(* Logix 5000 project; controller Amvex_Thorpe_Flowmeter vendor 1 type 14 code 106 rev 33.13; software revision 33.01; part 9 of 16 *)

ADD_ON_INSTRUCTION SetVelControlTimeOut   (* revision 0.1, vendor Mecademic Inc., ExecuteEnableInFalse *)
// Timeout for current velocity mode
VAR_IN_OUT
   RobotInputs : _061D:Meca500_86BDA20B:I:0; {required}
   RobotOutputs : _061D:Meca500_01F88326:O:0; {required}
END_VAR
VAR_INPUT
   Parameter_Value : REAL; {required}
   ExternalStateControl : BOOL; {required}
   ExternalMoveID : INT; {required}
END_VAR
VAR_OUTPUT
   Enabled : BOOL; {visible}
   Sent : BOOL; {visible}
   Buffered : BOOL; {visible}
   Error : BOOL; {visible}
END_VAR
VAR
   InternalMoveID : INT; {access None}
   MoveIDTrig : BOOL; {access None}
   MoveIDUpdated : BOOL; {access None}
   OneShot : DINT; {access None}
   FirstScan : BOOL; {access None}
END_VAR

ROUTINE EnableInFalse   (* ladder *)
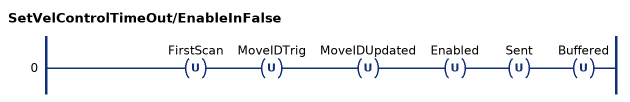
   0: OTU(FirstScan)OTU(MoveIDTrig)OTU(MoveIDUpdated)OTU(Enabled)OTU(Sent)OTU(Buffered);
END_ROUTINE

ROUTINE Logic   (* ladder *)
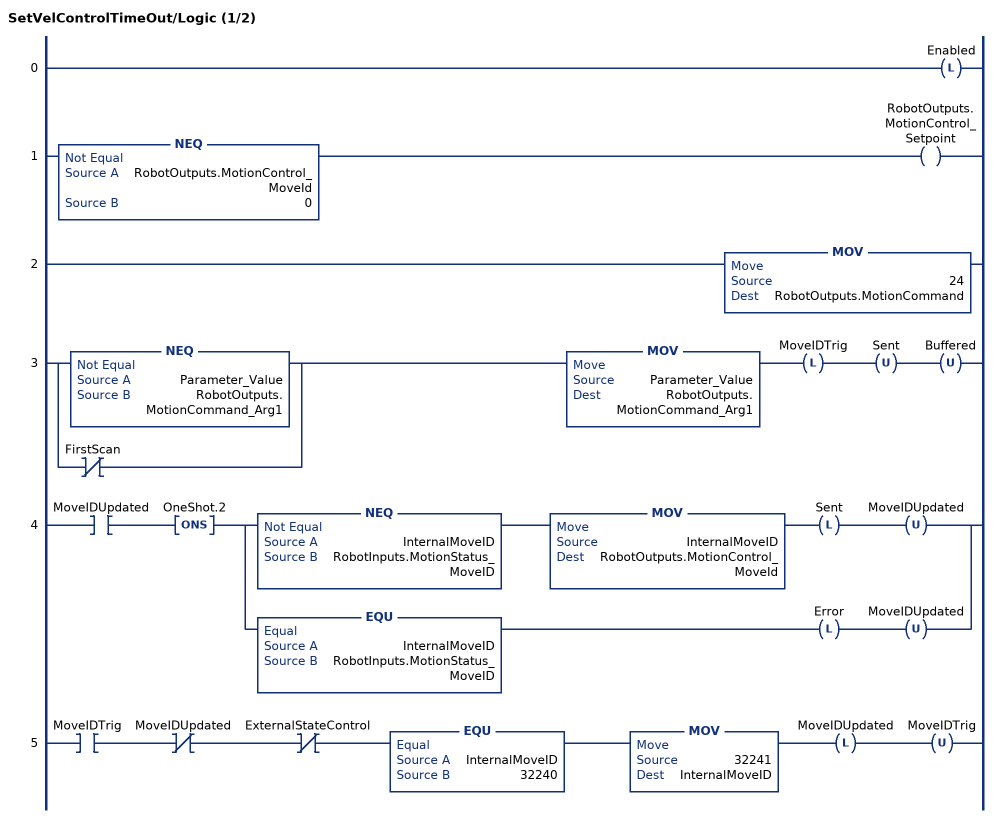
   0: OTL(Enabled);
   1: NEQ(RobotOutputs.MotionControl_MoveId,0)OTE(RobotOutputs.MotionControl_Setpoint);
   2: MOV(24,RobotOutputs.MotionCommand);
   3: [NEQ(Parameter_Value,RobotOutputs.MotionCommand_Arg1) ,XIO(FirstScan) ]MOV(Parameter_Value,RobotOutputs.MotionCommand_Arg1)OTL(MoveIDTrig)OTU(Sent)OTU(Buffered);
   4: XIC(MoveIDUpdated)ONS(OneShot.2)[NEQ(InternalMoveID,RobotInputs.MotionStatus_MoveID) MOV(InternalMoveID,RobotOutputs.MotionControl_MoveId) OTL(Sent) OTU(MoveIDUpdated) ,EQU(InternalMoveID,RobotInputs.MotionStatus_MoveID) OTL(Error) OTU(MoveIDUpdated) ];
   5: XIC(MoveIDTrig)XIO(MoveIDUpdated)XIO(ExternalStateControl)EQU(InternalMoveID,32240)MOV(32241,InternalMoveID)OTL(MoveIDUpdated)OTU(MoveIDTrig);
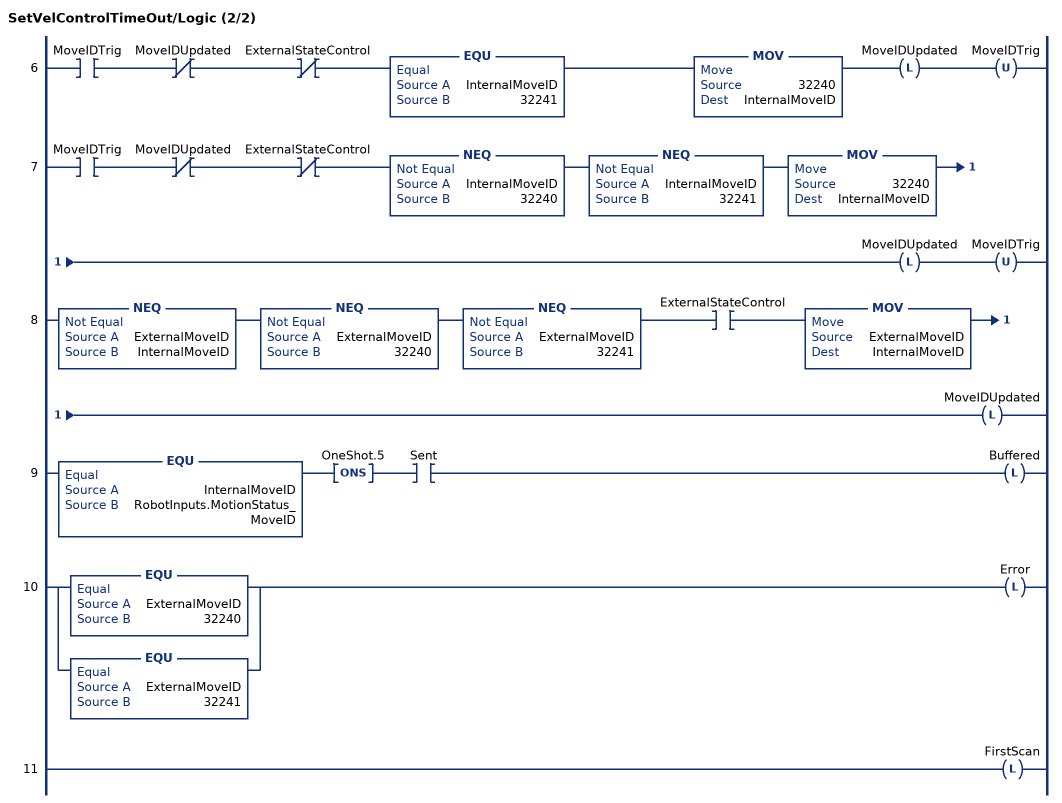
   6: XIC(MoveIDTrig)XIO(MoveIDUpdated)XIO(ExternalStateControl)EQU(InternalMoveID,32241)MOV(32240,InternalMoveID)OTL(MoveIDUpdated)OTU(MoveIDTrig);
   7: XIC(MoveIDTrig)XIO(MoveIDUpdated)XIO(ExternalStateControl)NEQ(InternalMoveID,32240)NEQ(InternalMoveID,32241)MOV(32240,InternalMoveID)OTL(MoveIDUpdated)OTU(MoveIDTrig);
   8: NEQ(ExternalMoveID,InternalMoveID)NEQ(ExternalMoveID,32240)NEQ(ExternalMoveID,32241)XIC(ExternalStateControl)MOV(ExternalMoveID,InternalMoveID)OTL(MoveIDUpdated);
   9: EQU(InternalMoveID,RobotInputs.MotionStatus_MoveID)ONS(OneShot.5)XIC(Sent)OTL(Buffered);
   10: [EQU(ExternalMoveID,32240) ,EQU(ExternalMoveID,32241) ]OTL(Error);
   11: OTL(FirstScan);
END_ROUTINE
END_ADD_ON_INSTRUCTION

ADD_ON_INSTRUCTION SetWRF   (* revision 0.1, vendor Mecademic Inc., ExecuteEnableInFalse *)
// Set the pose of the WRF with respect of the BRF
VAR_IN_OUT
   RobotInputs : _061D:Meca500_86BDA20B:I:0; {required}
   RobotOutputs : _061D:Meca500_01F88326:O:0; {required}
END_VAR
VAR_INPUT
   Pose_X_Pos : REAL; {required}
   Pose_Y_Pos : REAL; {required}
   Pose_Z_Pos : REAL; {required}
   Pose_rX_Ang : REAL; {required}
   Pose_rY_Ang : REAL; {required}
   Pose_rZ_Ang : REAL; {required}
   ExternalStateControl : BOOL; {required}
   ExternalMoveID : INT; {required}
END_VAR
VAR_OUTPUT
   Enabled : BOOL; {visible}
   Sent : BOOL; {visible}
   Buffered : BOOL; {visible}
   Error : BOOL; {visible}
END_VAR
VAR
   InternalMoveID : INT; {access None}
   MoveIDTrig : BOOL; {access None}
   MoveIDUpdated : BOOL; {access None}
   OneShot : DINT; {access None}
   FirstScan : BOOL; {access None}
END_VAR

ROUTINE EnableInFalse   (* ladder *)
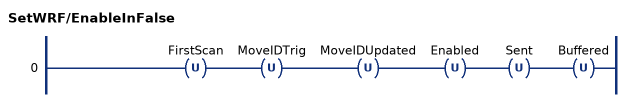
   0: OTU(FirstScan)OTU(MoveIDTrig)OTU(MoveIDUpdated)OTU(Enabled)OTU(Sent)OTU(Buffered);
END_ROUTINE

ROUTINE Logic   (* ladder *)
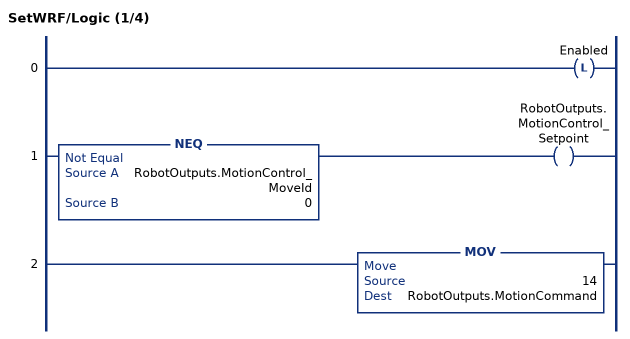
   0: OTL(Enabled);
   1: NEQ(RobotOutputs.MotionControl_MoveId,0)OTE(RobotOutputs.MotionControl_Setpoint);
   2: MOV(14,RobotOutputs.MotionCommand);
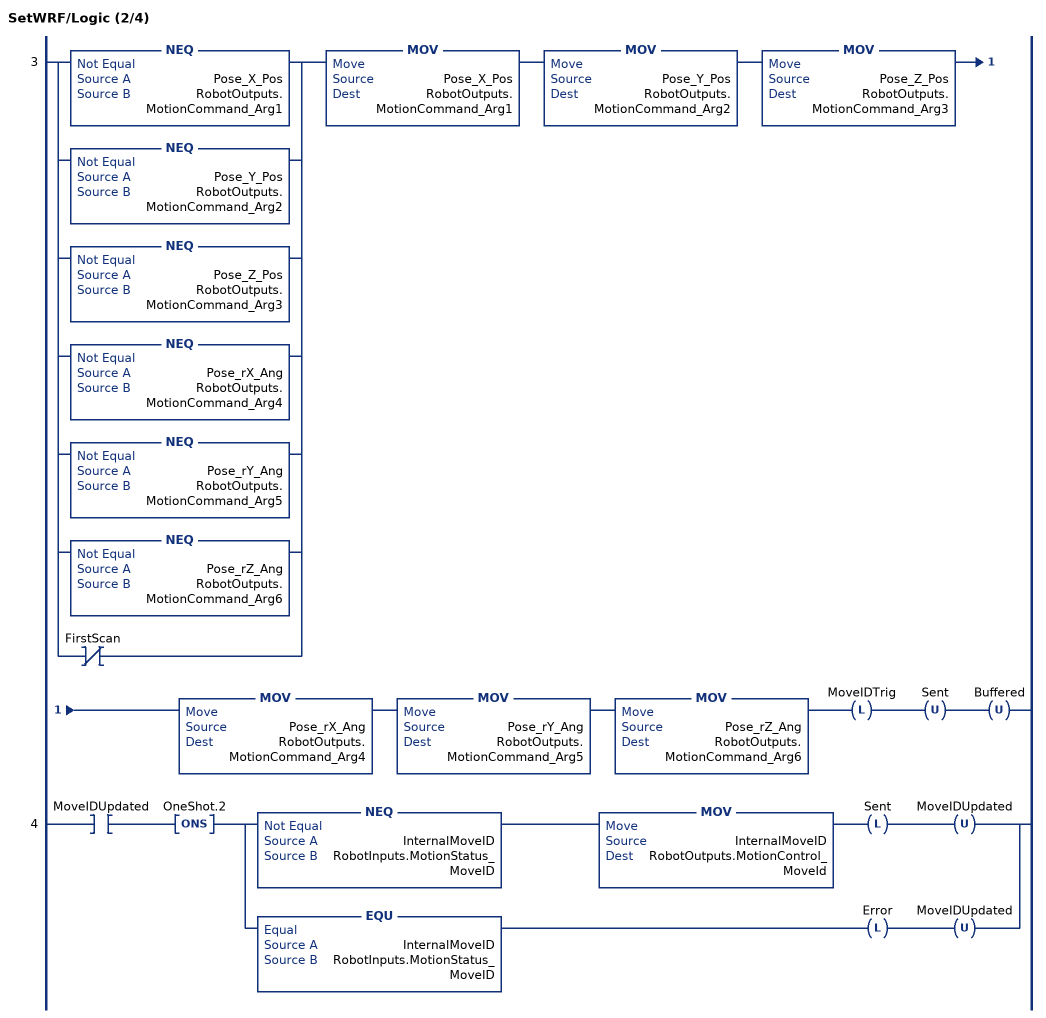
   3: [NEQ(Pose_X_Pos,RobotOutputs.MotionCommand_Arg1) ,NEQ(Pose_Y_Pos,RobotOutputs.MotionCommand_Arg2) ,NEQ(Pose_Z_Pos,RobotOutputs.MotionCommand_Arg3) ,NEQ(Pose_rX_Ang,RobotOutputs.MotionCommand_Arg4) ,NEQ(Pose_rY_Ang,RobotOutputs.MotionCommand_Arg5) ,NEQ(Pose_rZ_Ang,RobotOutputs.MotionCommand_Arg6) ,XIO(FirstScan) ]MOV(Pose_X_Pos,RobotOutputs.MotionCommand_Arg1)MOV(Pose_Y_Pos,RobotOutputs.MotionCommand_Arg2)MOV(Pose_Z_Pos,RobotOutputs.MotionCommand_Arg3)MOV(Pose_rX_Ang,RobotOutputs.MotionCommand_Arg4)MOV(Pose_rY_Ang,RobotOutputs.MotionCommand_Arg5)MOV(Pose_rZ_Ang,RobotOutputs.MotionCommand_Arg6)OTL(MoveIDTrig)OTU(Sent)OTU(Buffered);
   4: XIC(MoveIDUpdated)ONS(OneShot.2)[NEQ(InternalMoveID,RobotInputs.MotionStatus_MoveID) MOV(InternalMoveID,RobotOutputs.MotionControl_MoveId) OTL(Sent) OTU(MoveIDUpdated) ,EQU(InternalMoveID,RobotInputs.MotionStatus_MoveID) OTL(Error) OTU(MoveIDUpdated) ];
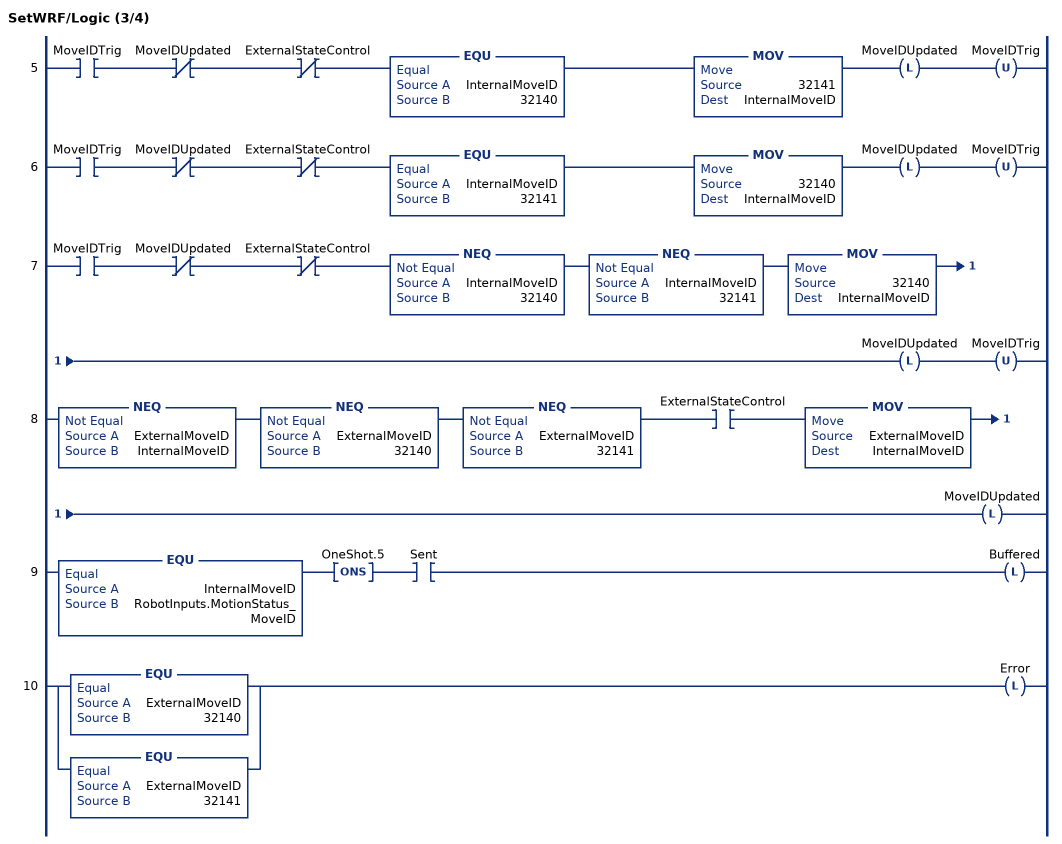
   5: XIC(MoveIDTrig)XIO(MoveIDUpdated)XIO(ExternalStateControl)EQU(InternalMoveID,32140)MOV(32141,InternalMoveID)OTL(MoveIDUpdated)OTU(MoveIDTrig);
   6: XIC(MoveIDTrig)XIO(MoveIDUpdated)XIO(ExternalStateControl)EQU(InternalMoveID,32141)MOV(32140,InternalMoveID)OTL(MoveIDUpdated)OTU(MoveIDTrig);
   7: XIC(MoveIDTrig)XIO(MoveIDUpdated)XIO(ExternalStateControl)NEQ(InternalMoveID,32140)NEQ(InternalMoveID,32141)MOV(32140,InternalMoveID)OTL(MoveIDUpdated)OTU(MoveIDTrig);
   8: NEQ(ExternalMoveID,InternalMoveID)NEQ(ExternalMoveID,32140)NEQ(ExternalMoveID,32141)XIC(ExternalStateControl)MOV(ExternalMoveID,InternalMoveID)OTL(MoveIDUpdated);
   9: EQU(InternalMoveID,RobotInputs.MotionStatus_MoveID)ONS(OneShot.5)XIC(Sent)OTL(Buffered);
   10: [EQU(ExternalMoveID,32140) ,EQU(ExternalMoveID,32141) ]OTL(Error);
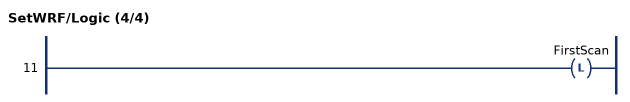
   11: OTL(FirstScan);
END_ROUTINE
END_ADD_ON_INSTRUCTION

ADD_ON_INSTRUCTION StartOfflineProgram   (* revision 0.1, vendor Mecademic Inc., ExecuteEnableInFalse *)
// Start an offline program with specified id
VAR_IN_OUT
   RobotInputs : _061D:Meca500_86BDA20B:I:0; {required}
   RobotOutputs : _061D:Meca500_01F88326:O:0; {required}
END_VAR
VAR_INPUT
   Parameter_Value : REAL; {required}
   ExternalStateControl : BOOL; {required}
   ExternalMoveID : INT; {required}
END_VAR
VAR_OUTPUT
   Enabled : BOOL; {visible}
   Sent : BOOL; {visible}
   Buffered : BOOL; {visible}
   Error : BOOL; {visible}
END_VAR
VAR
   InternalMoveID : INT; {access None}
   MoveIDTrig : BOOL; {access None}
   MoveIDUpdated : BOOL; {access None}
   OneShot : DINT; {access None}
   FirstScan : BOOL; {access None}
END_VAR

ROUTINE EnableInFalse   (* ladder *)
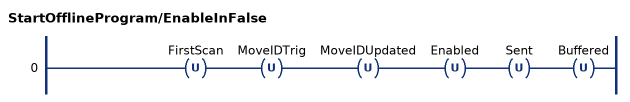
   0: OTU(FirstScan)OTU(MoveIDTrig)OTU(MoveIDUpdated)OTU(Enabled)OTU(Sent)OTU(Buffered);
END_ROUTINE

ROUTINE Logic   (* ladder *)
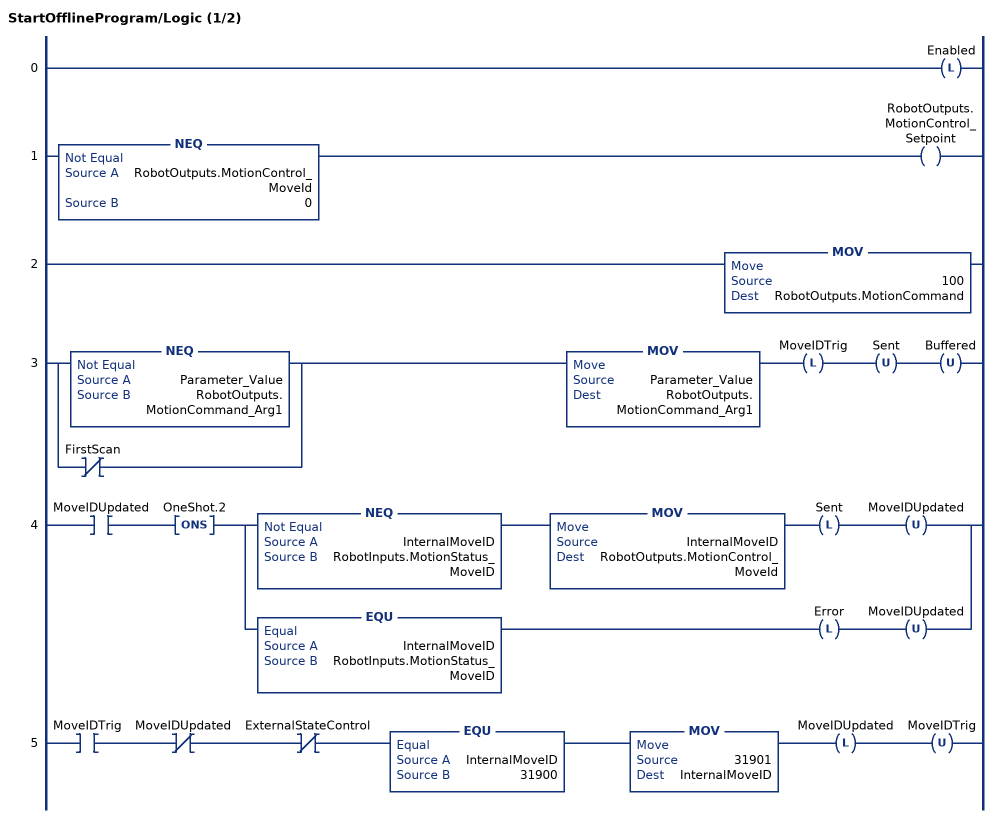
   0: OTL(Enabled);
   1: NEQ(RobotOutputs.MotionControl_MoveId,0)OTE(RobotOutputs.MotionControl_Setpoint);
   2: MOV(100,RobotOutputs.MotionCommand);
   3: [NEQ(Parameter_Value,RobotOutputs.MotionCommand_Arg1) ,XIO(FirstScan) ]MOV(Parameter_Value,RobotOutputs.MotionCommand_Arg1)OTL(MoveIDTrig)OTU(Sent)OTU(Buffered);
   4: XIC(MoveIDUpdated)ONS(OneShot.2)[NEQ(InternalMoveID,RobotInputs.MotionStatus_MoveID) MOV(InternalMoveID,RobotOutputs.MotionControl_MoveId) OTL(Sent) OTU(MoveIDUpdated) ,EQU(InternalMoveID,RobotInputs.MotionStatus_MoveID) OTL(Error) OTU(MoveIDUpdated) ];
   5: XIC(MoveIDTrig)XIO(MoveIDUpdated)XIO(ExternalStateControl)EQU(InternalMoveID,31900)MOV(31901,InternalMoveID)OTL(MoveIDUpdated)OTU(MoveIDTrig);
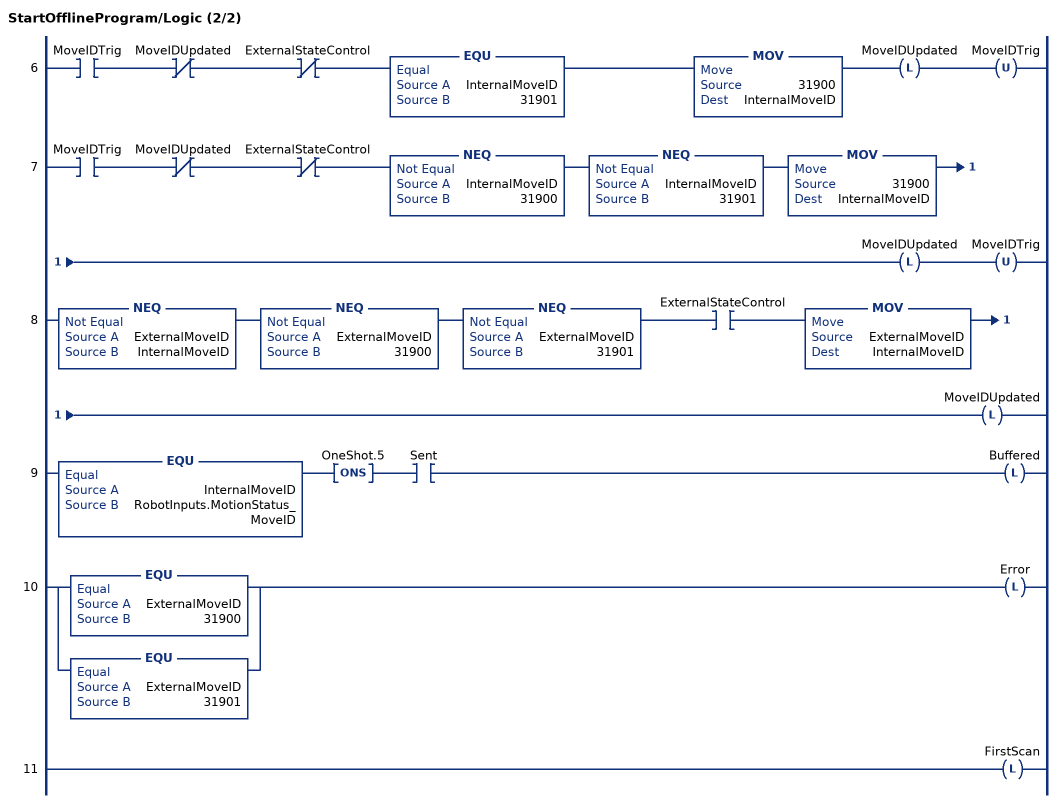
   6: XIC(MoveIDTrig)XIO(MoveIDUpdated)XIO(ExternalStateControl)EQU(InternalMoveID,31901)MOV(31900,InternalMoveID)OTL(MoveIDUpdated)OTU(MoveIDTrig);
   7: XIC(MoveIDTrig)XIO(MoveIDUpdated)XIO(ExternalStateControl)NEQ(InternalMoveID,31900)NEQ(InternalMoveID,31901)MOV(31900,InternalMoveID)OTL(MoveIDUpdated)OTU(MoveIDTrig);
   8: NEQ(ExternalMoveID,InternalMoveID)NEQ(ExternalMoveID,31900)NEQ(ExternalMoveID,31901)XIC(ExternalStateControl)MOV(ExternalMoveID,InternalMoveID)OTL(MoveIDUpdated);
   9: EQU(InternalMoveID,RobotInputs.MotionStatus_MoveID)ONS(OneShot.5)XIC(Sent)OTL(Buffered);
   10: [EQU(ExternalMoveID,31900) ,EQU(ExternalMoveID,31901) ]OTL(Error);
   11: OTL(FirstScan);
END_ROUTINE
END_ADD_ON_INSTRUCTION

VAR_GLOBAL   (* controller tags *)
   Air_Pressure_Issue_Delay_TMR : TIMER := (PRE := 1000, ACC := 1000, EN := 1, DN := 1);
   Alicat1RequestMsg : MESSAGE;
        MessageParameters(ServiceCode := 16#0010, LocalElement := MCP.Testing.Alicat[0].CmdData[0], ...)
   Alicat1ResponseMsg : MESSAGE;
        MessageParameters(ServiceCode := 16#000e, DestinationTag := MCP.Testing.Alicat[0].CmdData[0], ...)
   Alicat2RequestMsg : MESSAGE;
        MessageParameters(ServiceCode := 16#0010, LocalElement := MCP.Testing.Alicat[1].CmdData[0], ...)
   Alicat2ResponseMsg : MESSAGE;
        MessageParameters(ServiceCode := 16#000e, DestinationTag := MCP.Testing.Alicat[1].CmdData[0], ...)
   Alicat5LPM_Timeout : TIMER := (PRE := 3000);
   Alicat_Status_ONS : BOOL[32];
   Barcode_Data_String : STRING := '62810150300021T15UOB00032$0D$00$00$00$00$00$00$00$00$00$00$00$00$00$00$00$00$00$00$00$00$00$00$00$00$00$00$00$00$00$00$00$00$00$00$00$00$00$00$00$00$00$00$00$00$00$00$00$00$00$00$00$00$00$00$00$00$00$00';
   Barcode_Data_Temp : DINT;
   Barcode_Delay : TIMER := (PRE := 500);
   Barcode_timeout : TIMER := (PRE := 2000);
   Blank_Nest_Release_TMR : TIMER := (PRE := 500);
   Close : BOOL;
   Close_Go_ONS : BOOL;
   Close_Knob : Servo_Move := (Speed := 400.0, Torque := 37.0, Position := 100000.0, Path := 1);
   Close_Knob_Step : Servo_Move := (Speed := 600.0, Torque := 35.0, Position := -100000.0, Path := 1);
   Close_ONS : BOOL;
   Close_Rapid : Servo_Move := (Speed := 8000.0, Torque := 80.0, Position := 550000.0, Path := 1);
   Close_Step : Servo_Move := (Speed := 600.0, Torque := 37.0, Position := 1000000.0, Path := 1);
   Close_Stop : BOOL;
   Close_Torque : INT := 36;
   Close_Torque_TMR : TIMER;
   CloseKnob : Servo_Move := (Speed := 200.0, Torque := 55.0, Position := 1000000.0, Path := 1);
   Cycle_Count_Ctr : COUNTER := (ACC := 1765, DN := 1);
   Cycle_Count_ONS : BOOL;
   Cycle_Time_ONS : BOOL;
   Cycle_Timer_ONS : BOOL;
   Datalogging_Time_Delay : TIMER := (PRE := 500);
   Delay : TIMER := (PRE := 3000);
   Downsteam_Release_ONS1 : BOOL;
   Downsteam_Release_ONS2 : BOOL;
   Empty_Pallet_Timer : TIMER := (PRE := 5000);
   Empty_Pallet_Timer2 : TIMER := (PRE := 5000);
   End_Of_Cycle : BOOL;
   Fastest_Delay : TIMER := (PRE := 100);
   FIRST_SCAN : BOOL;
   FIRST_SCAN_ONS : BOOL := 1;
   Fitting_Cycle_Timer : TIMER := (PRE := 6000000);
   Fitting_Cycle_Timer_DINT : DINT;
   Fitting_Cycle_Timer_ONS : BOOL;
   Flood_delay : TIMER := (PRE := 10000, ACC := 10000, EN := 1, DN := 1);
   Flowmeter_Record : STRING;
   HMI : HMI_Temp;
   ID0_InputDataLength : MESSAGE;   // Message Command Input Data Data Length
        MessageParameters(ServiceCode := 16#000e, DestinationTag := RCP1_00.MISC.InputBytes, ...)
   ID0_LengthParameterdata : MESSAGE;   // Message Command Parameter Data Length
        MessageParameters(ServiceCode := 16#000e, DestinationTag := RCP1_00.MISC.ParameterBytes, ...)
   ID0_MSG_Diagnostic : MESSAGE;   // Message Get Diagnosis Module
        MessageParameters(ServiceCode := 16#000e, DestinationTag := RCP1_00.MISC.DiagnosticData[0], ...)
   ID0_MSG_ProcessAlarm : MESSAGE;   // Message Get Get Process Alram Module
        MessageParameters(ServiceCode := 16#000e, DestinationTag := RCP1_00.MISC.ProcessAlarmData[0], ...)
   ID0_OutputDataLength : MESSAGE;   // Message Command Output Data Data Length
        MessageParameters(ServiceCode := 16#000e, DestinationTag := RCP1_00.MISC.OutputBytes, ...)
   ID0_ReceiveMSG1 : MESSAGE;   // Message Command Parameter Receive Data
        MessageParameters(ServiceCode := 16#000e, DestinationTag := RCP1_00.MISC.ParameterArray_RX_TX[0], ...)
   ID0_ReceiveMSG2 : MESSAGE;   // Message Command Parameter Receive Data
        MessageParameters(ServiceCode := 16#000e, DestinationTag := RCP1_00.MISC.ParameterArray_RX_TX[450], ...)
   ID0_ReceiveMSG3 : MESSAGE;   // Message Command Parameter Receive Data
        MessageParameters(ServiceCode := 16#000e, DestinationTag := RCP1_00.MISC.ParameterArray_RX_TX[900], ...)
   ID0_SendMSG1 : MESSAGE;   // Message Command Parameter Send Data
        MessageParameters(ServiceCode := 16#0010, LocalElement := RCP1_00.MISC.ParameterArray_RX_TX[0], ...)
   ID0_SendMSG2 : MESSAGE;   // Message Command Parameter Send Data
        MessageParameters(ServiceCode := 16#0010, LocalElement := RCP1_00.MISC.ParameterArray_RX_TX[450], ...)
   ID0_SendMSG3 : MESSAGE;   // Message Command Parameter Send Data
        MessageParameters(ServiceCode := 16#0010, LocalElement := RCP1_00.MISC.ParameterArray_RX_TX[900], ...)
   ID86_InputDataLength : MESSAGE;   // Message Command Input Data Data Length
        MessageParameters(ServiceCode := 16#000e, DestinationTag := MCP_00.MISC.InputBytes, ...)
   ID86_LengthParameterdata : MESSAGE;   // Message Command Parameter Data Length
        MessageParameters(ServiceCode := 16#000e, DestinationTag := MCP_00.MISC.ParameterBytes, ...)
   ID86_MSG_Diagnostic : MESSAGE;   // Message Get Diagnosis Module
        MessageParameters(ServiceCode := 16#000e, DestinationTag := MCP_00.MISC.DiagnosticData[0], ...)
   ID86_MSG_ProcessAlarm : MESSAGE;   // Message Get Get Process Alram Module
        MessageParameters(ServiceCode := 16#000e, DestinationTag := MCP_00.MISC.ProcessAlarmData[0], ...)
   ID86_OutputDataLength : MESSAGE;   // Message Command Output Data Data Length
        MessageParameters(ServiceCode := 16#000e, DestinationTag := MCP_00.MISC.OutputBytes, ...)
   ID86_ReceiveMSG1 : MESSAGE;   // Message Command Parameter Receive Data
        MessageParameters(ServiceCode := 16#000e, DestinationTag := MCP_00.MISC.ParameterArray_RX_TX[0], ...)
   ID86_ReceiveMSG2 : MESSAGE;   // Message Command Parameter Receive Data
        MessageParameters(ServiceCode := 16#000e, DestinationTag := MCP_00.MISC.ParameterArray_RX_TX[450], ...)
   ID86_ReceiveMSG3 : MESSAGE;   // Message Command Parameter Receive Data
        MessageParameters(ServiceCode := 16#000e, DestinationTag := MCP_00.MISC.ParameterArray_RX_TX[900], ...)
   ID86_SendMSG1 : MESSAGE;   // Message Command Parameter Send Data
        MessageParameters(ServiceCode := 16#0010, LocalElement := MCP_00.MISC.ParameterArray_RX_TX[0], ...)
   ID86_SendMSG2 : MESSAGE;   // Message Command Parameter Send Data
        MessageParameters(ServiceCode := 16#0010, LocalElement := MCP_00.MISC.ParameterArray_RX_TX[450], ...)
   ID86_SendMSG3 : MESSAGE;   // Message Command Parameter Send Data
        MessageParameters(ServiceCode := 16#0010, LocalElement := MCP_00.MISC.ParameterArray_RX_TX[900], ...)
   In_Cycle : BOOL := 1;
   Job_Number : STRING;
   KB_DeBug : DINT := 8424448;
   KB_Temp_Ret_TM : TIMER := (PRE := 600, ACC := 600, EN := 1, DN := 1);
   Knob_Closer : Servo_Move := (Speed := 600.0, Torque := 37.0, Position := -100000.0, Path := 1);
   Knob_Servo_Reset : BOOL := 1;
   Knob_Temp_Seq_Start : BOOL;
   Knob_Turner_ONS : BOOL;
   Last_Test_Data : REAL[8] := ([1] := 0.0001953125, [2] := 6.9492188, [3] := 15.0859375, [4] := 52.21875, [5] := 0.0005859375);
   Load_PB_ONS : BOOL;
   MCP : MCP := (Conv.VFD.Speed := 400, Conv.VFD.Ready := 1, Conv.Stop[0].Present.INPUT := 1, Conv.Stop[0].Present.ON_TIME := 100.0, Conv.Stop[0].Present.OFF_TIME := 50.0, Conv.Stop[0].Present.DEB_INPUT := 1, Conv.Stop[0].Present.IN := 1, Conv.Stop[0].Present.OUT := 1, Conv.Stop[1].Present.ON_TIME := 50.0, Conv.Stop[1].Present.OFF_TIME := 50.0, Conv.Stop[2].Present.INPUT := 1, Conv.Stop[2].Present.ON_TIME := 100.0, Conv.Stop[2].Present.OFF_TIME := 50.0, Conv.Stop[2].Present.DEB_INPUT := 1, Conv.Stop[2].Present.IN := 1, Conv.Stop[2].Present.OUT := 1, Conv.Lift.Stop.Present.INPUT := 1, Conv.Lift.Stop.Present.ON_TIME := 100.0, Conv.Lift.Stop.Present.OFF_TIME := 50.0, Conv.Lift.Stop.Present.DEB_INPUT := 1, Conv.Lift.Stop.Present.IN := 1, Conv.Lift.Stop.Present.OUT := 1, Conv.Lift.Extd.INPUT := 1, Conv.Lift.Extd.ON_TIME := 100.0, Conv.Lift.Extd.OFF_TIME := 50.0, Conv.Lift.Extd.DEB_INPUT := 1, Conv.Lift.Extd.IN := 1, Conv.Lift.Extd.OUT := 1, Conv.Lift.Retd.ON_TIME := 100.0, Conv.Lift.Retd.OFF_TIME := 50.0, Conv.Drop_TM[0].PRE := 250, Conv.Downstream_Full.ON_TIME := 50.0, Conv.Downstream_Full.OFF_TIME := 1000.0, Conv.Reject_Full.INPUT := 1, Conv.Reject_Full.ON_TIME := 250.0, Conv.Reject_Full.OFF_TIME := 50.0, Conv.Reject_Full.DEB_INPUT := 1, Conv.Reject_Full.IN := 1, Conv.Reject_Full.OUT := 1, Testing.Robot.Connection.Connect := 1, Testing.Robot.Connection.ConnectionFailed := 1, Testing.Robot.Lin_Speed := 85.0, Testing.Robot.Turn_TM.PRE := 350, Testing.Robot.Turn_Speed := 75.0, Testing.Robot.Turn_ONS := 1, Testing.Robot.MoveLin_Pos[0] := 64.35501, Testing.Robot.MoveLin_Pos[1] := 90.0, Testing.Robot.MoveLin_Pos[2] := 358.12, Testing.Robot.MoveLin_Pos[3] := -90.128174, Testing.Robot.MoveLin_Pos[4] := 2.1866865e-07, Testing.Robot.MoveLin_Pos[5] := -29.132236, Testing.Robot.Tool_Position_1[0] := 64.35501, Testing.Robot.Tool_Position_1[1] := 90.0, Testing.Robot.Tool_Position_1[2] := 358.12, Testing.Robot.Tool_Position_1[3] := -90.128174, Testing.Robot.Tool_Position_1[4] := 2.1866865e-07, Testing.Robot.Tool_Position_1[5] := -29.132236, Testing.Robot.Tool_Position_2[0] := 64.355, Testing.Robot.Tool_Position_2[1] := 130.0, Testing.Robot.Tool_Position_2[2] := 358.12,
        Testing.Robot.Tool_Position_2[3] := -90.0, Testing.Robot.Tool_Position_2[4] := -4.4799222e-07, Testing.Robot.Tool_Position_2[5] := -34.710915, Testing.Robot.At_Pos_1 := 1, Testing.Robot.DN := 1, Testing.Robot.Knob_Torque := 50.0, Testing.Robot.Jog.Increment := 5.0, Testing.Robot.Turn_Speed_AOI.Parameter_Value := 75.0, Testing.Robot.Turn_AOI.Joint_1_Angle := 17.26414, Testing.Robot.Turn_AOI.Joint_2_Angle := -8.834411, Testing.Robot.Turn_AOI.Joint_3_Angle := -19.158821, Testing.Robot.Turn_AOI.Joint_4_Angle := -98.415184, Testing.Robot.Turn_AOI.Joint_5_Angle := -74.87032, Testing.Robot.Torque_Config_AOI.Severity := 2.0, Testing.Robot.Torque_Limit_AOI.Joint_1_Limit := 100.0, Testing.Robot.Torque_Limit_AOI.Joint_2_Limit := 100.0, Testing.Robot.Torque_Limit_AOI.Joint_3_Limit := 100.0, Testing.Robot.Torque_Limit_AOI.Joint_4_Limit := 100.0, Testing.Robot.Torque_Limit_AOI.Joint_5_Limit := 100.0, Testing.Robot.Torque_Limit_AOI.Joint_6_Limit := 50.0, Testing.Robot.MoveLin_AOI.Pose_X_Pos := 64.35501, Testing.Robot.MoveLin_AOI.Pose_Y_Pos := 90.0, Testing.Robot.MoveLin_AOI.Pose_Z_Pos := 358.12, Testing.Robot.MoveLin_AOI.Pose_rX_Ang := -90.128174, Testing.Robot.MoveLin_AOI.Pose_rY_Ang := 2.1866865e-07, Testing.Robot.MoveLin_AOI.Pose_rZ_Ang := -29.132236, Testing.Robot.LinVel_AOI.Parameter_Value := 85.0, Testing.Robot.Open := 1, Testing.FastTest.Extd.INPUT := 1, Testing.FastTest.Extd.ON_TIME := 100.0, Testing.FastTest.Extd.OFF_TIME := 50.0, Testing.FastTest.Extd.DEB_INPUT := 1, Testing.FastTest.Extd.IN := 1, Testing.FastTest.Extd.OUT := 1, Testing.FastTest.Retd.ON_TIME := 100.0, Testing.FastTest.Retd.OFF_TIME := 50.0, Testing.Hood.Extd.INPUT := 1, Testing.Hood.Extd.ON_TIME := 100.0, Testing.Hood.Extd.OFF_TIME := 50.0, Testing.Hood.Extd.DEB_INPUT := 1, Testing.Hood.Extd.IN := 1, Testing.Hood.Extd.OUT := 1, Testing.Hood.Retd.ON_TIME := 100.0, Testing.Hood.Retd.OFF_TIME := 50.0, Testing.Alicat[0].IoData.Pressure := 14.396875, Testing.Alicat[0].IoData.Temperature := 28.3375, Testing.Alicat[0].IoData.VolFlow := 0.0001953125, Testing.Alicat[0].IoData.MassFlow := 0.0001953125, Testing.Alicat[0].IoData.GasIndex := 11, Testing.Alicat[0].IoData.Config := 16#0f, Testing.Alicat[0].IoData.PRESS := 1, Testing.Alicat[0].IoData.TEMP := 1, Testing.Alicat[0].IoData.VFLOW := 1, Testing.Alicat[0].IoData.MFLOW := 1, Testing.Alicat[0].Oxygen.To_100LPM := 1, Testing.Alicat[0].Ready := 1, Testing.Alicat[0].Flow := 0.0001953125, Testing.Alicat[0].Flow_data[0] := 1.5392579, Testing.Alicat[0].Flow_data[1] := 1.5396484, Testing.Alicat[0].Flow_data[2] := 1.5369141,
        Testing.Alicat[0].Flow_data[3] := 1.5371094, Testing.Alicat[0].Flow_data[4] := 1.5373048, Testing.Alicat[0].Flow_data[5] := 1.5378907, Testing.Alicat[0].Flow_data[6] := 1.5378907, Testing.Alicat[0].Flow_data[7] := 1.5382813, Testing.Alicat[0].Flow_data[8] := 1.5386719, Testing.Alicat[0].Flow_data[9] := 1.5386719, Testing.Alicat[0].Flow_data[10] := 1.5388672, Testing.Alicat[0].Flow_TM1.PRE := 1000, Testing.Alicat[0].Flow_TM2.PRE := 75, Testing.Alicat[1].IoData.Pressure := 14.396094, Testing.Alicat[1].IoData.Temperature := 25.284376, Testing.Alicat[1].IoData.VolFlow := 0.00390625, Testing.Alicat[1].IoData.MassFlow := 0.00390625, Testing.Alicat[1].IoData.GasIndex := 11, Testing.Alicat[1].IoData.Config := 16#0f, Testing.Alicat[1].IoData.PRESS := 1, Testing.Alicat[1].IoData.TEMP := 1, Testing.Alicat[1].IoData.VFLOW := 1, Testing.Alicat[1].IoData.MFLOW := 1, Testing.Alicat[1].Ready := 1, Testing.Alicat[1].Flow := 0.00390625, Testing.Alicat[1].Flow_data[0] := 7.8242188, Testing.Alicat[1].Flow_data[1] := 7.8164062, Testing.Alicat[1].Flow_data[2] := 7.8085938, Testing.Alicat[1].Flow_data[3] := 7.8046875, Testing.Alicat[1].Flow_data[4] := 7.796875, Testing.Alicat[1].Flow_data[5] := 7.796875, Testing.Alicat[1].Flow_data[6] := 7.796875, Testing.Alicat[1].Flow_data[7] := 7.84375, Testing.Alicat[1].Flow_data[8] := 7.8476562, Testing.Alicat[1].Flow_data[9] := 7.8398438, Testing.Alicat[1].Flow_data[10] := 7.8320312, Testing.Alicat[1].Flow_TM1.PRE := 1000, Testing.Alicat[1].Flow_TM2.PRE := 75, Testing.Alicat[1].Upper_Lim_Num := 8.8, Testing.Alicat[1].Lower_Lim_Num := 7.2, Testing.Vision.Prog := 3, Testing.Vision.Current_Prog := 3, Testing.Vision.Trigger_ON_TM.PRE := 33, Testing.Vision.Trigger_OFF_TM.PRE := 33, Testing.Barcode.Ready := 1, Testing.Barcode.Result := '010062810150300021T15UOB00032$0D', Testing.Part_Present.ON_TIME := 500.0, Testing.Part_Present.OFF_TIME := 50.0, Testing.Saftey.Light_Curtain := 1, Testing.Saftey.Output := 1, Testing.Saftey.RDC_Code := 15332, Testing.Air_pressure.INPUT := 1, Testing.Air_pressure.ON_TIME := 100.0, Testing.Air_pressure.OFF_TIME := 50.0, Testing.Air_pressure.DEB_INPUT := 1, Testing.Air_pressure.IN := 1, Testing.Air_pressure.OUT := 1, Testing.Part[39].Code := '010062810150300021T15UOB35098$0D', Testing.Part[39].Results := 56, Testing.Test[1].Range := 0.1, Testing.Test[1].Test_TM.PRE := 500, Testing.Test[1].Time := 1000, Testing.Test[2].Flow := 2.0,
        Testing.Test[2].Range := 0.5, Testing.Test[2].Test_TM.PRE := 500, Testing.Test[2].Time := 50, Testing.Test[3].Flow := 8.0, Testing.Test[3].Range := 0.8, Testing.Test[3].Test_TM.PRE := 500, Testing.Test[3].Time := 1, Testing.Test[4].Flow := 15.0, Testing.Test[4].Range := 1.5, Testing.Test[4].Test_TM.PRE := 500, Testing.Test[4].Time := 4007, Testing.Test[5].Flow := 50.0, Testing.Test[5].Range := 20.0, Testing.Test[5].Test_TM.PRE := 500, Testing.Test[5].Time := 13, Testing.Test[6].Test_TM.PRE := 1000, Testing.Test[6].Time := 4884, Testing.Load_PB.ON_TIME := 50.0, Testing.Load_PB.OFF_TIME := 50.0, Testing.Knob_Turner.Enable := 1, Testing.Knob_Turner.Stop := 1, Testing.Knob_Turner.Turn_Speed := 50.0, Testing.Knob_Turner.Rapid_Speed := 600.0, Testing.Knob_Turner.T2_Rapid_Pos := 550000.0, Testing.Knob_Turner.Torque_EN1 := 1, Testing.Knob_Turner.Torque_Feedback := 3.0, Testing.Knob_Turner.Path := 1.0, Testing.Knob_Turner.Extd.INPUT := 1, Testing.Knob_Turner.Extd.ON_TIME := 50.0, Testing.Knob_Turner.Extd.OFF_TIME := 50.0, Testing.Knob_Turner.Extd.DEB_INPUT := 1, Testing.Knob_Turner.Extd.IN := 1, Testing.Knob_Turner.Extd.OUT := 1, Testing.Knob_Turner.Retd.ON_TIME := 100.0, Testing.Knob_Turner.Retd.OFF_TIME := 50.0, Part_Count := 98, Lifetime_Part_Count := 5720.0, Fault_AOI[0].Timer_PRE := 2500, Fault_AOI[1].Timer_PRE := 2500, Fault_AOI[2].Timer_PRE := 2500, Fault_AOI[3].Timer_PRE := 2500, Fault_AOI[4].Timer_PRE := 2500, Fault_AOI[5].Timer_PRE := 2500, Fault_AOI[6].Timer_PRE := 2500, Fault_AOI[7].Timer_PRE := 2500, Fault_AOI[8].Timer_PRE := 2500, Fault_AOI[9].Timer_PRE := 2500, Fault_AOI[10].Timer_PRE := 2500, Fault_AOI[11].Timer_PRE := 2500, Fault_AOI[12].Timer_PRE := 2500, Fault_AOI[13].Timer_PRE := 2500, Fault_AOI[14].Timer_PRE := 2500, Fault_AOI[15].Timer_PRE := 2500, Fault_AOI[16].Timer_PRE := 2500, Fault_AOI[17].Timer_PRE := 2500, Fault_AOI[18].Timer_PRE := 2500, Fault_AOI[19].Timer_PRE := 2500, Fault_AOI[20].Timer_PRE := 2500, Fault_AOI[21].Fault := 1, Fault_AOI[21].Bypass := 1,
        Fault_AOI[21].Timer_PRE := 13, Fault_AOI[21].Faulted := 1, Fault_AOI[22].Fault := 1, Fault_AOI[22].Timer_PRE := 63968020, Fault_AOI[22].Timer_ACC := 4079810, Fault_AOI[23].Timer_PRE := 11, Fault_AOI[23].Timer_ACC := 483196928, Fault_AOI[24].Fault := 1, Fault_AOI[24].Bypass := 1, Fault_AOI[25].Timer_PRE := 1330795077, Fault_AOI[25].Timer_ACC := 808464688, Fault_AOI[26].Timer_PRE := 1112495413, Fault_AOI[26].Timer_ACC := 858796080, Fault_AOI[26].Faulted := 1, Fault_AOI[26].Reset := 1, Fault_AOI[29].Fault := 1, Fault_AOI[29].Timer_PRE := 1112014848, Fault_AOI[29].Timer_ACC := 1112014848, Fault_AOI[29].Faulted := 1, Fault_AOI[29].Reset := 1, Fault_AOI[30].Fault := 1, Fault_AOI[30].Bypass := 1, Fault_AOI[30].Timer_PRE := 50, Fault_AOI[30].Timer_ACC := 50, Fault_AOI[31].Fault := 1, Fault_AOI[31].Bypass := 1, Fault_AOI[31].Timer_PRE := 4210882, Fault_AOI[31].Timer_ACC := 1, Fault_AOI[31].Faulted := 1, Fault[0] := 1111490560, Fault[1] := 1112014848, Performance := 8315.151, Availability := inf, UptimeSTM.PRE := 60000, UptimeM.PRE := 60, DowntimeSTM.PRE := 6000, DowntimeSTM.ACC := 6000, DowntimeSTM.EN := 1, DowntimeSTM.DN := 1, DowntimeM.PRE := 60, DowntimeM.ACC := 24, Cycle_Time := 28, UptimeH.ACC := 3, UptimeH.DN := 1, DowntimeH.ACC := 12, DowntimeH.DN := 1, UptimeTM.PRE := 1000, DowntimeTM.PRE := 1000, UptimeS.PRE := 60, UptimeS.ACC := 33, DowntimeS.PRE := 60, DowntimeS.ACC := 17, HMI.Conv.VFD.Speed := 40, HMI.Conv.Stop[0].Present.INPUT := 1, HMI.Conv.Stop[0].Present.ON_TIME := 4.36e-43, HMI.Conv.Stop[0].Present.OFF_TIME := 50.0, HMI.Conv.Stop[0].Present.DEB_INPUT := 1, HMI.Conv.Stop[1].Present.ON_TIME := -1.7e-44, HMI.Conv.Stop[1].Present.OFF_TIME := -9.1766204e+29, HMI.Conv.Stop[1].Present.DEB_INPUT := 1,
        HMI.Conv.Stop[1].Present.ON_TT := 1, HMI.Conv.Stop[2].Present.ON_TIME := 9.745e-41, HMI.Conv.Stop[2].Present.OFF_TIME := 7.e-44, HMI.Conv.Stop[3].Present.RESET := 1, HMI.Conv.Stop[3].Present.ON_TIME := -4.2e-44, HMI.Conv.Stop[3].Present.OFF_TIME := -9.1766204e+29, HMI.Conv.Stop[3].Release := 1, HMI.Conv.Stop[3].Hold := 1, HMI.Conv.Stop[4].Present.ON_TIME := 2.7301833e+23, HMI.Conv.Stop[4].Present.OFF_TIME := -107613980.0, HMI.Conv.Lift.Stop.Present.ON_TIME := 3.528607e+09, HMI.Conv.Lift.Stop.Present.OFF_TIME := 6.4098327e-10, HMI.Conv.Diverter.Present.INPUT := 1, HMI.Conv.Diverter.Present.RESET := 1, HMI.Conv.Diverter.Present.ON_TIME := 7.e-44, HMI.Conv.Diverter.Present.OFF_TIME := 7.e-44, HMI.Conv.Diverter.Present.OFF_TT := 1, HMI.Conv.Drop_TM[0].PRE := 3, HMI.Conv.Drop_TM[0].ACC := 311, HMI.Conv.Drop_TM[1].PRE := 1112014848, HMI.Conv.Drop_TM[1].ACC := 69543, HMI.Conv.Drop_TM[1].TT := 1, HMI.Conv.Drop_TM[2].ACC := -1325330291, HMI.Testing.Robot.Connection.ConnectionInhibited := 1, HMI.Testing.Robot.Connection.ConnectionFailed := 1, HMI.Testing.Robot.Setup := 8, HMI.Testing.Robot.Lin_Speed := -4.2e-44, HMI.Testing.Robot.Unturn := 1, HMI.Testing.Robot.Turn_TM.PRE := 4079810, HMI.Testing.Robot.Turn_TM.ACC := 1, HMI.Testing.Robot.Turn_Deg := 3.9e-44, HMI.Testing.Robot.Turn_Speed := 4.e-45, HMI.Testing.Robot.MoveLin_Pos[0] := 1.5e-44, HMI.Testing.Robot.MoveLin_Pos[1] := 1.3565762e-21, HMI.Testing.Robot.MoveLin_Pos[2] := 2.7301833e+23, HMI.Testing.Robot.MoveLin_Pos[3] := -107613980.0, HMI.Testing.Robot.MoveLin_Pos[4] := -107858530.0, HMI.Testing.Robot.MoveLin_Pos[5] := 6.6472e-41, HMI.Testing.Robot.Tool_Position_2[0] := 3.528607e+09, HMI.Testing.Robot.Tool_Position_2[1] := 6.4098327e-10, HMI.Testing.Robot.Tool_Position_2[2] := 2.6804066e-09, HMI.Testing.Robot.Tool_Position_2[3] := 6.5917316e-10, HMI.Testing.Robot.Tool_Position_2[4] := 6.409692e-10, HMI.Testing.Robot.Tool_Position_2[5] := 3.0878025e-09, HMI.Testing.Robot.To_Pos_1 := 1, HMI.Testing.Robot.At_Pos_1 := 1, HMI.Testing.Robot.Pos_1_Set := 1, HMI.Testing.Robot.Pos_2_Set := 1, HMI.Testing.Robot.Pause := 1, HMI.Testing.Robot.Knob_Torque := 4.102202e-08, HMI.Testing.Robot.Jog.Enabled := 1, HMI.Testing.Robot.Jog.X_Inc := 2.8e-44, HMI.Testing.Robot.Jog.Y_Inc := 4.36e-43, HMI.Testing.Robot.Jog.Z_Inc := 50.0, HMI.Testing.Robot.Jog.Increment := 50.0, HMI.Testing.Robot.Jog.Speed := 9.4703e-41, HMI.Testing.Robot.Turn_Speed_AOI.ExternalMoveID := 4236, HMI.Testing.Robot.Turn_Speed_AOI.Sent := 1, HMI.Testing.Robot.Turn_Speed_AOI.Buffered := 1, HMI.Testing.Robot.Turn_AOI.Joint_1_Angle := -1.12e-43,
        HMI.Testing.Robot.Turn_AOI.Joint_2_Angle := -1.7e-44, HMI.Testing.Robot.Turn_AOI.Joint_3_Angle := -9.1766204e+29, HMI.Testing.Robot.Turn_AOI.Joint_4_Angle := 1.2229299e-36, HMI.Testing.Robot.Turn_AOI.Joint_5_Angle := 5.900702e-39, HMI.Testing.Robot.Turn_AOI.Joint_6_Angle := 1.e-45, HMI.Testing.Robot.Turn_AOI.Sent := 1, HMI.Testing.Robot.Turn_AOI.Buffered := 1, HMI.Testing.Robot.ErrorAOI.CommandBufferFull := 1, HMI.Testing.Robot.ErrorAOI.SyntaxError := 1, HMI.Testing.Robot.ErrorAOI.ArgumentError := 1, HMI.Testing.Robot.ErrorAOI.JointOverLimit := 1, HMI.Testing.Robot.Torque_Config_AOI.Severity := 9.745e-41, HMI.Testing.Robot.Torque_Config_AOI.Detection_Mode := 7.e-44, HMI.Testing.Robot.Torque_Limit_AOI.Joint_1_Limit := 3.08e-43, HMI.Testing.Robot.Torque_Limit_AOI.Joint_2_Limit := 1.8e-44, HMI.Testing.Robot.Torque_Limit_AOI.Joint_5_Limit := -1.1e-44, HMI.Testing.Robot.Torque_Limit_AOI.Joint_6_Limit := -4.2e-44, HMI.Testing.Robot.Torque_Limit_AOI.ExternalMoveID := 20996, HMI.Testing.Robot.Torque_Limit_AOI.Sent := 1, HMI.Testing.Robot.Torque_Limit_AOI.Buffered := 1, HMI.Testing.Robot.MoveLin_AOI.Pose_X_Pos := 1.e-45, HMI.Testing.Robot.MoveLin_AOI.Pose_Y_Pos := 3.9e-44, HMI.Testing.Robot.MoveLin_AOI.Pose_Z_Pos := 4.e-45, HMI.Testing.Robot.MoveLin_AOI.Pose_rY_Ang := 1.5e-44, HMI.Testing.Robot.MoveLin_AOI.Pose_rZ_Ang := 1.3565762e-21, HMI.Testing.Robot.MoveLin_AOI.ExternalMoveID := 16746, HMI.Testing.Robot.MoveLin_AOI.Error := 1, HMI.Testing.Robot.LinVel_AOI.Parameter_Value := 6.6472e-41, HMI.Testing.Robot.LinVel_AOI.ExternalStateControl := 1, HMI.Testing.Robot.LinVel_AOI.Enabled := 1, HMI.Testing.Robot.LinVel_AOI.Error := 1, HMI.Testing.Robot.Open := 1, HMI.Testing.FastTest.Extd.OFF_TIME := 3.528607e+09, HMI.Testing.FastTest.Retd.ON_TIME := 4.732e-42, HMI.Testing.FastTest.Retd.DEB_INPUT := 1, HMI.Testing.FastTest.Retd.IN := 1, HMI.Testing.Hood.Retd.INPUT := 1, HMI.Testing.Hood.Retd.RESET := 1, HMI.Testing.Hood.Retd.ON_TIME := 7.e-44, HMI.Testing.Hood.Retd.DEB_INPUT := 1, HMI.Testing.Hood.Retd.IN := 1, HMI.Testing.Hood.Retd.ON_TT := 1, HMI.Testing.Hood.Retd.OFF_TT := 1, HMI.Testing.Hood.Retd.OUT := 1, HMI.Testing.Alicat[0].Test := 1, HMI.Testing.Alicat[0].CMD_AOI.CmdResult := 3, HMI.Testing.Alicat[0].CMD_AOI.START := 1, HMI.Testing.Alicat[0].IoData.Status := 16#0000_0032, HMI.Testing.Alicat[0].IoData.T_UNDR := 1, HMI.Testing.Alicat[0].IoData.M_OVER := 1, HMI.Testing.Alicat[0].IoData.M_UNDR := 1, HMI.Testing.Alicat[0].IoData.Temperature := -1.8781379e-09, HMI.Testing.Alicat[0].IoData.VolFlow := 7.e-44, HMI.Testing.Alicat[0].IoData.MassFlow := 3.08e-43, HMI.Testing.Alicat[0].IoData.ActualSetpoint := 1.8e-44, HMI.Testing.Alicat[0].IoData.RequestedSetpoint := -1.1e-44, HMI.Testing.Alicat[0].IoData.GasIndex := 30, HMI.Testing.Alicat[0].CmdData[0] := 20996, HMI.Testing.Alicat[0].CmdData[1] := -3783, HMI.Testing.Alicat[0].Oxygen.To_100LPM := 1,
        HMI.Testing.Alicat[0].Oxygen.To_5LPM := 1, HMI.Testing.Alicat[0].Flow := 1.e-45, HMI.Testing.Alicat[0].Flow_Avg := 3.9e-44, HMI.Testing.Alicat[0].Flow_data[0] := 4.e-45, HMI.Testing.Alicat[0].Flow_data[2] := 1.5e-44, HMI.Testing.Alicat[0].Flow_data[3] := 1.3565762e-21, HMI.Testing.Alicat[0].Flow_data[4] := 2.7301833e+23, HMI.Testing.Alicat[0].Flow_data[5] := -107613980.0, HMI.Testing.Alicat[0].Flow_data[6] := -107858530.0, HMI.Testing.Alicat[0].Flow_data[7] := 6.6472e-41, HMI.Testing.Alicat[0].Flow_data[14] := 3.528607e+09, HMI.Testing.Alicat[0].Flow_data[15] := 6.4098327e-10, HMI.Testing.Alicat[0].Flow_data[16] := 2.6804066e-09, HMI.Testing.Alicat[0].Flow_data[17] := 6.5917316e-10, HMI.Testing.Alicat[0].Flow_data[18] := 6.409692e-10, HMI.Testing.Alicat[0].Flow_data[19] := 3.0878025e-09, HMI.Testing.Alicat[0].Flow_data[20] := 51.83321, HMI.Testing.Alicat[0].Flow_data[21] := 4.102202e-08, HMI.Testing.Alicat[0].Flow_data[22] := 4.732e-42, HMI.Testing.Alicat[1].IoData.Status := 16#0001_07fe, HMI.Testing.Alicat[1].IoData.T_UNDR := 1, HMI.Testing.Alicat[1].IoData.V_OVER := 1, HMI.Testing.Alicat[1].IoData.V_UNDR := 1, HMI.Testing.Alicat[1].IoData.M_OVER := 1, HMI.Testing.Alicat[1].IoData.M_UNDR := 1, HMI.Testing.Alicat[1].IoData.P_OVER := 1, HMI.Testing.Alicat[1].IoData.TOT_OVER := 1, HMI.Testing.Alicat[1].IoData.HLD := 1, HMI.Testing.Alicat[1].IoData.ADC := 1, HMI.Testing.Alicat[1].IoData.EXH := 1, HMI.Testing.Alicat[1].IoData.Pressure := 7.e-44, HMI.Testing.Alicat[1].IoData.VolFlow := -1.09322e-19, HMI.Testing.Alicat[1].IoData.MassFlow := 7.e-44, HMI.Testing.Alicat[1].IoData.ActualSetpoint := 7.e-44, HMI.Testing.Alicat[1].IoData.ValveDrivePct := -1.12e-43, HMI.Testing.Alicat[1].IoData.Totalizer := -1.7e-44, HMI.Testing.Alicat[1].IoData.RequestedSetpoint := -9.1766204e+29, HMI.Testing.Alicat[1].IoData.GasIndex := 4636, HMI.Testing.Alicat[1].IoData.Config := 16#d0, HMI.Testing.Alicat[1].IoData.SP := 1, HMI.Testing.Alicat[1].IoData.TOTAL := 1, HMI.Testing.Alicat[1].CmdData[0] := 16578, HMI.Testing.Alicat[1].CmdData[1] := 64, HMI.Testing.Alicat[1].Oxygen.Oxygen := 1, HMI.Testing.Alicat[1].Flow := 4.e-45, HMI.Testing.Alicat[1].Flow_Avg := 4.36e-43, HMI.Testing.Alicat[1].Flow_data[0] := 50.0, HMI.Testing.Alicat[1].Flow_data[1] := 50.0, HMI.Testing.Alicat[1].Flow_data[2] := 9.745e-41, HMI.Testing.Alicat[1].Flow_data[3] := 7.e-44, HMI.Testing.Alicat[1].Flow_data[5] := -1.8781379e-09, HMI.Testing.Alicat[1].Flow_data[6] := 7.e-44, HMI.Testing.Alicat[1].Flow_data[7] := 3.08e-43, HMI.Testing.Alicat[1].Flow_data[8] := 1.8e-44, HMI.Testing.Alicat[1].Flow_data[11] := -1.1e-44, HMI.Testing.Alicat[1].Flow_data[12] := -4.2e-44, HMI.Testing.Alicat[1].Flow_data[13] := -9.1766204e+29, HMI.Testing.Alicat[1].Flow_data[14] := 1.2229521e-36, HMI.Testing.Alicat[1].Flow_data[15] := 5.717031e-39, HMI.Testing.Alicat[1].Flow_data[16] := 1.e-45,
        HMI.Testing.Alicat[1].Flow_data[17] := 3.9e-44, HMI.Testing.Alicat[1].Flow_data[18] := 4.e-45, HMI.Testing.Alicat[1].Flow_data[20] := 1.5e-44, HMI.Testing.Alicat[1].Flow_data[21] := 1.3565762e-21, HMI.Testing.Alicat[1].Flow_data[22] := 2.7301833e+23, HMI.Testing.Alicat[1].Flow_data[23] := -107613980.0, HMI.Testing.Alicat[1].Flow_data[24] := -107858530.0, HMI.Testing.Vision.Enable := 1, HMI.Testing.Vision.Result_OK := 1, HMI.Testing.Vision.Busy := 1, HMI.Testing.Vision.Prog := 82, HMI.Testing.Vision.Current_Prog := 82, HMI.Testing.Vision.Trigger_ON_TM.PRE := 825766454, HMI.Testing.Vision.Trigger_ON_TM.ACC := 808792368, HMI.Testing.Vision.Trigger_ON_TM.DN := 1, HMI.Testing.Vision.Trigger_OFF_TM.PRE := 827601202, HMI.Testing.Vision.Trigger_OFF_TM.ACC := 1112495413, HMI.Testing.Vision.Trigger_OFF_TM.DN := 1, HMI.Testing.Barcode.Result := '$00$00$00$00$00$00$00$00$00$00$00$00$00$00$00$00$00$00$00$00$00$00$00$00$00$00$00$00$00$00$00$00$00$00$00$00$00$00$00$00$00$00$00$00$00$00$00$00$00$00$00$00$14$00$00$007$01$00$00$00$00HB$00$00HB$FE$07$01$002$00$00$00$00$00$00$00$8C$10$01$A0', HMI.Testing.Barcode.Result_avalible := 1, HMI.Testing.Barcode.Read_success := 1, HMI.Testing.Barcode.Read_failed := 1, HMI.Testing.Part_Present.ON_TIME := -1.12e-43, HMI.Testing.Part_Present.OFF_TIME := -1.7e-44, HMI.Testing.Part_Present.DEB_INPUT := 1, HMI.Testing.Part_Present.IN := 1, HMI.Testing.Saftey.Lockout := 1, HMI.Testing.Saftey.Input_Fault := 1, HMI.Testing.Saftey.Output_Fault := 1, HMI.Testing.Saftey.Light_Curtain := 1, HMI.Testing.Saftey.Door := 1, HMI.Testing.Saftey.RDC_Active := 1, HMI.Testing.Air_pressure.INPUT := 1, HMI.Testing.Air_pressure.RESET := 1, HMI.Testing.Air_pressure.ON_TIME := 1.8e-44, HMI.Testing.Air_pressure.DEB_INPUT := 1, HMI.Testing.Air_pressure.ON_TT := 1, HMI.Testing.Air_pressure.OFF_TT := 1, HMI.Testing.Stacklight.Green := 1, HMI.Testing.Part[0].Code := '$03$00$00$00$00$00$00$00$0B$00$00$00$00$00$CD$1CjAgf$E4A$CD$CCL$B9$CD$CC', HMI.Testing.Part[0].Results := 12336, HMI.Testing.Part[1].Code := '$00$00$00$00$00$00$00$00$00$00$00$00$00$00$00$00$00$00$00$00$00$00$00$00$00$00$00$00$00$00$00$00$00$00$00$00$00$00$00$00$00$00$00$00$00$00$00$00$00$00$00$00$14$00$00$007$01$00$00$00$00HB$00$00HB$FE$07$01$002$00$00$00$00$00$00$00$8C$10$01$A0', HMI.Testing.Part[1].Results := 50, HMI.Testing.Part[2].Code := 'P$00$00$80$0C$00$00$80$04R9$F1$1C$12$D0$03$C2@@$00$01$00$00$00$00$00$00$00$03$00$00$007$01$00$00$00$00HB$00$00HB$A7$0F$01$002$00', HMI.Testing.Part[2].Results := 30, HMI.Testing.Part[3].Code := '$14$13$D0$03$C2@>$00$01$00$00$00$1C$00$00$00$03$00$00$00$00$00$00$00$0B$00$00$00$00$00$CD$1CjAgf$E4A$CD$CCL$B9$CD$CCL$B9$00$00$00$00$00$00$00$00$00$00$00$00$00$00$00$00$00$00$00$00$00$00$00$00$00$00ERRO01006281', HMI.Testing.Part[3].Results := 12592, HMI.Testing.Part[4].Code := '21T15UOB00031$0D$00$00$00$00$00$00$00$00$00$00$00$00$00$00$00$00$00$00$00$00$00$00$00$00$00$00$00$00$00$00$00$00$00$00$00$00$00$00$00$00$00$00$00$00$00$00$00$00$00$00$00$00$00$00$14$00$00$007$01$00$00$00$00HB$00$00HB', HMI.Testing.Part[4].Results := 2046, HMI.Testing.Part[5].Code := '$00$00$00$00$8C$10$01$A02$00$00$002$00$00$00P$00$00$80$0C$00$00$80$04R9$F1$1C$12$D0$03$C2@@$00$01$00$00$00$00$00$00$00$03$00$00$007$01', HMI.Testing.Part[5].Results := 13, HMI.Testing.Part[7].Code := '010062810150300021T15UOB00031$0D$00$00$00$00$00$00$00$00$00$00$00$00$00$00$00$00$00$00$00$00$00$00$00$00$00$00$00$00$00$00$00$00$00$00$00$00$00$00$00$00$00$00$00$00$00$00$00$00$00$00$00$00$00$00', HMI.Testing.Part[7].Results := 20, HMI.Testing.Part[8].Code := '$00$00HB$00$00HB$FE$07$01$002$00$00$00$00$00$00$00$8C$10$01$A02$00$00$002$00$00$00P$00$00$80$0C$00$00$80$04R9$F1$1C$12$D0$03$C2@@$00$01$00$00$00$00$00$00$00$03$00$00$007$01$00$00$00$00HB$00$00HB$A7$0F$01$002$00$00$00', HMI.Testing.Part[9].Code := '2$00$00$00$DC$00$00$00$0D$00$00$00$00$00$00$00$00$00$00$00$08$00$00$80$1E$00$00$80$04R9$F1$14$13$D0$03$C2@>$00$01$00$00$00$1C$00$00$00$03$00$00$00$00$00$00$00$0B$00$00$00$00$00$CD$1CjAgf$E4A$CD$CCL$B9$CD$CCL$B9$00$00$00$00$00$00', HMI.Testing.Part[12].Code := '$A7$0F$01$002$00$00$00$00$00$00$00$8D$10$01$B12$00$00$00$DC$00$00$00$0D$00$00$00$00$00$00$00$00$00$00$00$08$00$00$80$1E$00$00$80$04R9$F1$14$13$D0$03$C2@>$00$01$00$00$00$1C$00$00$00$03$00$00$00$00$00$00$00$0B$00$00$00$00$00$CD$1CjAgf', HMI.Testing.Part[12].Results := 16868, HMI.Testing.Part[13].Code := 'L$B9$00$00$00$00$00$00$00$00$00$00$00$00$00$00$00$00$00$00$00$00$00$00$00$00$00$00ERRO010062810150300021T15UOB00031$0D$00$00$00$00$00$00$00$00$00$00$00$00$00$00$00$00$00$00$00$00$00$00', HMI.Testing.Part[14].Results := 1, HMI.Testing.Part[16].Code := '$00$00$CD$1CjAgf$E4A$CD',
        HMI.Testing.Part[17].Results := 12, HMI.Testing.Part[18].Code := '$1C$12$D0$03$C2@@$00$01$00$00$00$00$00$00$00$03$00$00$007$01$00$00$00$00HB$00$00HB$A7$0F$01$002$00$00$00$00$00$00$00$8D$10$01$B12$00$00$00$DC$00$00$00$0D$00$00$00$00$00$00$00$00$00$00$00$08$00$00$80$1E$00$00$80$04R9$F1$14$13$D0$03', HMI.Testing.Part[18].Results := 16578, HMI.Testing.Part[19].Code := '$1C', HMI.Testing.Part[19].Results := 21813, HMI.Testing.Part[20].Code := '1$0D$00$00$00$00$00$00$00$00$00$00$00$00$00$00$00$00$00$00$00$00$00$00$00$00$00$00$00$00$00$00$00$00$00$00$00$00$00$00$00$00$00$00$00$00$00$00$00$00$00$00$00$00$00$00$14$00$00$007$01$00$00$00$00HB$00$00HB$FE$07$01$002$00$00$00$00$00$00$00', HMI.Testing.Part[20].Results := 4236, HMI.Testing.Part[21].Code := '2$00$00$00P$00$00$80$0C$00$00$80$04R9$F1$1C$12$D0$03$C2@@$00$01$00$00$00$00$00$00$00$03$00$00$007$01$00$00$00$00HB$00$00HB$A7$0F', HMI.Testing.Part[21].Results := 8, HMI.Testing.Part[22].Code := '$04R9$F1$14$13$D0$03$C2@>$00$01$00$00$00$1C$00$00$00$03$00$00$00$00$00$00$00$0B$00$00$00$00$00$CD$1CjAgf$E4A$CD$CCL$B9$CD$CCL$B9$00$00$00$00$00$00$00$00$00$00$00$00$00$00$00$00$00$00$00$00$00$00$00$00$00$00ERRO0100', HMI.Testing.Part[22].Results := 12854, HMI.Testing.Part[23].Code := '300021T15UOB00031$0D$00$00$00$00$00$00$00$00$00$00$00$00$00$00$00$00$00$00$00$00$00$00$00$00$00$00$00$00$00$00$00$00$00$00$00$00$00$00$00$00$00$00$00$00$00$00$00$00$00$00$00$00$00$00$14$00$00$007$01$00$00$00$00HB', HMI.Testing.Part[24].Code := '2$00$00$00$00$00$00$00$8C$10$01$A02$00$00$002$00$00$00P$00$00$80$0C$00$00$80$04R9$F1$1C$12$D0$03$C2@@$00$01$00$00$00$00$00$00$00$03$00$00$007$01$00$00$00$00HB$00$00HB$A7$0F$01$002$00$00$00$00$00$00$00$8D$10$01$B12$00$00$00', HMI.Testing.Part[24].Results := 220, HMI.Testing.Part[25].Code := '$00$00$00$00$00$00$00$00$08$00$00$80$1E', HMI.Testing.Part[27].Code := '7$01$00$00$00$00HB$00$00HB$FE$07$01$002$00$00$00', HMI.Testing.Part[27].Results := 50, HMI.Testing.Part[30].Results := 311, HMI.Testing.Part[31].Code := '$00$00HB$A7$0F$01$002$00$00$00$00$00$00$00$8D$10$01$B12$00$00$00$DC$00$00$00$0D$00$00$00$00$00$00$00$00$00$00$00$08$00$00$80$1E$00$00$80$04R9$F1$14$13$D0$03$C2@>$00$01$00$00$00$1C$00$00$00$03$00$00$00$00$00$00$00$0B$00$00$00$00$00$CD$1C', HMI.Testing.Part[31].Results := 16746, HMI.Testing.Part[32].Code := 'L$B9$CD$CCL$B9$00$00$00$00$00$00$00$00$00$00$00$00$00$00$00$00$00$00$00$00$00$00$00$00$00$00ERRO010062810150300021T15UOB00031$0D$00$00$00$00$00$00$00$00$00$00$00$00$00$00$00$00$00$00', HMI.Testing.Part[33].Results := 16578, HMI.Testing.Part[34].Results := 3, HMI.Testing.Part[36].Results := 80, HMI.Testing.Part[37].Code := '$04R9$F1$1C$12$D0$03$C2@@$00$01$00$00$00$00$00$00$00$03$00$00$007$01$00$00$00$00HB$00$00HB$A7$0F$01$002$00$00$00$00$00$00$00$8D$10$01$B12$00$00$00$DC$00$00$00$0D$00$00$00$00$00$00$00$00$00$00$00$08$00$00$80$1E$00$00$80$04R9$F1', HMI.Testing.Part[37].Results := 4884, HMI.Testing.Part[38].Code := '$01$00$00$00$1C$00$00$00$03$00$00$00$00$00$00$00$0B$00$00$00$00$00$CD$1CjAgf$E4A$CD$CCL$B9$CD$CCL$B9$00$00$00$00$00$00$00$00$00$00$00$00$00$00$00$00$00$00$00$00$00$00$00$00$00$00ERRO0100628101503000', HMI.Testing.Part[38].Results := 12594, HMI.Testing.Part[39].Code := '00031$0D$00$00$00$00$00$00$00$00$00$00$00$00$00$00$00$00$00$00$00$00$00$00$00$00$00$00$00$00$00$00$00$00$00$00$00$00$00$00$00$00$00$00$00$00$00$00$00$00$00$00$00$00$00$00$14$00$00$007$01$00$00$00$00HB$00$00HB$FE$07$01$002$00$00$00', HMI.Testing.Part[40].Code := '2$00$00$002$00$00$00P$00$00$80$0C$00$00$80$04R9$F1$1C$12$D0$03$C2@@$00$01$00$00$00$00$00$00$00$03$00$00$007$01$00$00$00$00HB$00$00HB$A7$0F$01$002$00$00$00$00$00$00$00$8D$10$01$B12$00$00$00$DC$00$00$00$0D$00$00$00$00$00$00$00', HMI.Testing.Part[41].Code := '$1E$00$00$80$04R9$F1$14$13$D0$03$C2@>$00$01$00$00$00$1C$00$00$00$03$00$00$00$00$00$00$00$0B$00$00$00$00$00$CD$1CjAgf$E4A$CD$CCL$B9$CD$CCL$B9$00$00$00$00$00$00$00$00$00$00$00$00$00$00$00$00$00$00$00$00$00$00$00$00$00$00ERRO', HMI.Testing.Part[41].Results := 12592, HMI.Testing.Part[42].Code := '0150300021T15UOB00031$0D$00$00$00$00$00$00$00$00$00$00$00$00$00$00$00$00$00$00$00$00$00$00$00$00$00$00$00$00$00$00$00$00$00$00$00$00$00$00$00$00$00$00$00$00$00$00$00$00$00$00$00$00$00$00$14$00$00$007$01$00$00', HMI.Testing.Part[43].Code := '$FE$07$01$002$00$00$00$00$00$00$00$8C$10$01$A02$00$00$002$00$00$00P$00$00$80$0C$00$00$80$04R9$F1$1C$12$D0$03$C2@@$00$01$00$00$00$00$00$00$00$03$00$00$007$01$00$00$00$00HB$00$00HB$A7$0F$01$002$00$00$00$00$00$00$00$8D$10$01$B1', HMI.Testing.Part[43].Results := 50, HMI.Testing.Part[44].Code := '$0D$00$00$00$00$00$00$00$00$00$00$00$08$00$00$80$1E$00$00$80$04R9$F1$14$13$D0$03$C2@>$00$01$00$00$00$1C$00$00$00$03$00$00$00$00$00$00$00$0B$00$00$00$00$00$CD$1CjAgf$E4A$CD$CCL$B9$CD$CCL$B9$00$00$00$00$00$00$00$00$00$00$00$00$00$00', HMI.Testing.Part[46].Results := 4007, HMI.Testing.Part[47].Code := '$00$00$00$00$8D$10$01$B12$00$00$00$DC$00$00$00$0D$00$00$00$00$00$00$00$00$00$00$00$08$00$00$80$1E$00$00$80$04R9$F1$14$13$D0$03$C2@>$00$01$00', HMI.Testing.Part[47].Results := -18100, HMI.Testing.Part[49].Results := 3, HMI.Testing.Part[50].Code := '$00$00HB$00$00HB$A7$0F$01$002$00$00$00$00$00$00$00$8D$10$01$B12$00$00$00$DC$00$00$00$0D$00$00$00$00$00$00$00$00$00$00$00$08$00$00$80$1E$00$00$80$04R9$F1$14$13$D0$03$C2@>$00$01$00$00$00$1C$00$00$00$03$00$00$00$00$00$00$00$0B$00$00$00', HMI.Testing.Part[51].Code := '$E4A$CD$CCL$B9$CD$CCL$B9$00$00$00$00$00$00$00$00$00$00$00$00$00$00$00$00$00$00$00$00$00$00$00$00$00$00ERRO010062810150300021T15UOB00031$0D$00$00$00$00$00$00$00$00$00$00$00$00$00$00', HMI.Testing.Part[52].Results := 4636, HMI.Testing.Part[53].Code := '$01$00$00$00$00$00$00$00$03$00$00$007$01$00$00$00$00HB$00$00HB$A7$0F$01$002$00$00$00$00$00$00$00$8D$10$01$B12$00$00$00$DC$00$00$00$0D$00$00$00$00$00$00$00$00$00$00$00$08$00$00$80$1E$00$00$80$04R9$F1$14$13$D0$03$C2@>$00$01$00$00$00', HMI.Testing.Part[53].Results := 28, HMI.Testing.Part[54].Results := 3377, HMI.Testing.Part[55].Results := 50, HMI.Testing.Part[56].Code := '$0C$00$00$80$04R9$F1$1C$12$D0$03$C2@@$00$01$00$00$00$00$00$00$00$03$00$00$007$01$00$00$00$00HB$00$00HB$A7$0F$01$002$00$00$00$00$00$00$00$8D$10$01$B12$00$00$00$DC$00$00$00$0D$00$00$00$00$00$00$00$00$00$00$00$08$00$00$80$1E$00$00$80', HMI.Testing.Part[56].Results := 20996, HMI.Testing.Part[57].Code := '$C2@>$00$01$00$00$00$1C$00$00$00$03$00$00$00$00$00$00$00$0B$00$00$00$00$00$CD$1CjAgf$E4A$CD$CCL$B9$CD$CCL$B9$00$00$00$00$00$00$00$00$00$00$00$00$00$00$00$00$00$00$00$00$00$00$00$00$00$00ERRO010062810150', HMI.Testing.Part[57].Results := 12339, HMI.Testing.Part[58].Code := '5UOB00031$0D$00$00$00$00$00$00$00$00$00$00$00$00$00$00$00$00$00$00$00$00$00$00$00$00$00$00$00$00$00$00$00$00$00$00$00$00$00$00$00$00$00$00$00$00$00$00$00$00$00$00$00$00$00$00$14$00$00$007$01$00$00$00$00HB$00$00HB$FE$07$01$00', HMI.Testing.Part[58].Results := 50, HMI.Testing.Part[60].Results := 21061, HMI.Testing.Part[61].Code := '62810150300021T15UOB00031$0D$00$00$00$00$00$00$00$00$00$00$00$00$00$00$00$00$00$00$00$00$00$00$00$00$00$00$00$00$00$00$00$00$00$00$00$00$00$00$00$00$00$00$00$00$00$00$00$00$00$00$00$00$00$00$14$00$00$00', HMI.Testing.Part[61].Results := 311, HMI.Testing.Part[62].Code := '$00$00HB$FE$07$01$002$00$00$00$00$00$00$00$8C$10$01$A02$00$00$002$00$00$00P$00$00$80$0C$00$00$80$04R9$F1$1C$12$D0$03$C2@@$00$01$00$00$00$00$00$00$00$03$00$00$007$01$00$00$00$00HB$00$00HB$A7$0F$01$002$00$00$00$00$00$00$00', HMI.Testing.Part[62].Results := 4237, HMI.Testing.Part[63].Code := '$DC$00$00$00$0D$00$00$00$00$00$00$00$00$00$00$00$08$00$00$80$1E$00$00$80$04R9$F1$14$13$D0$03$C2@>$00$01$00$00$00$1C$00$00$00$03$00$00$00$00$00', HMI.Testing.Part[66].Code := '2$00$00$00$00$00$00$00$8D$10$01$B12$00$00$00$DC$00$00$00$0D$00$00$00$00$00$00$00$00$00$00$00$08$00$00$80$1E$00$00$80$04R9$F1$14$13$D0$03$C2@>$00$01$00$00$00$1C$00$00$00$03$00$00$00$00$00$00$00$0B$00$00$00$00$00$CD$1CjAgf$E4A$CD$CC',
        HMI.Testing.Part[66].Results := -18100, HMI.Testing.Part[67].Code := '$00$00$00$00$00$00$00$00$00$00$00$00$00$00$00$00$00$00$00$00$00$00$00$00ERRO010062810150300021T15UOB00031$0D$00$00$00$00$00$00$00$00$00$00$00$00$00$00$00$00$00$00$00$00$00$00$00$00$00$00', HMI.Testing.Part[69].Code := '7$01$00', HMI.Testing.Part[69].Results := 11, HMI.Testing.Part[70].Code := 'jAgf$E4A$CD$CCL$B9$CD$CCL$B9$00$00$00$00$00$00$00$00$00$00$00$00$00$00$00$00$00$00$00$00$00$00$00$00$00$00ERRO010062810150300021T15UOB00031$0D$00$00$00$00$00$00$00$00$00$00', HMI.Testing.Part[71].Results := 20996, HMI.Testing.Part[72].Code := '$C2@@$00$01$00$00$00$00$00$00$00$03$00$00$007$01$00$00$00$00HB$00$00HB$A7$0F$01$002$00$00$00$00$00$00$00$8D$10$01$B12$00$00$00$DC$00$00$00$0D$00$00$00$00$00$00$00$00$00$00$00$08$00$00$80$1E$00$00$80$04R9$F1$14$13$D0$03$C2@>$00', HMI.Testing.Part[72].Results := 1, HMI.Testing.Part[73].Code := '$03$00$00$00$00$00$00$00$0B$00$00$00$00$00$CD$1CjAgf$E4A$CD$CCL$B9$CD$CC', HMI.Testing.Part[73].Results := 12336, HMI.Testing.Part[74].Code := '$00$00$00$00$00$00$00$00$00$00$00$00$00$00$00$00$00$00$00$00$00$00$00$00$00$00$00$00$00$00$00$00$00$00$00$00$00$00$00$00$00$00$00$00$00$00$00$00$00$00$00$00$14$00$00$007$01$00$00$00$00HB$00$00HB$FE$07$01$002$00$00$00$00$00$00$00$8C$10$01$A0', HMI.Testing.Part[74].Results := 50, HMI.Testing.Part[75].Code := 'P$00$00$80$0C$00$00$80$04R9$F1$1C$12$D0$03$C2@@$00$01$00$00$00$00$00$00$00$03$00$00$007$01$00$00$00$00HB$00$00HB$A7$0F$01$002$00', HMI.Testing.Part[75].Results := 30, HMI.Testing.Part[76].Code := '$14$13$D0$03$C2@>$00$01$00$00$00$1C$00$00$00$03$00$00$00$00$00$00$00$0B$00$00$00$00$00$CD$1CjAgf$E4A$CD$CCL$B9$CD$CCL$B9$00$00$00$00$00$00$00$00$00$00$00$00$00$00$00$00$00$00$00$00$00$00$00$00$00$00ERRO01006281', HMI.Testing.Part[76].Results := 12592, HMI.Testing.Part[77].Code := '21T15UOB00031$0D$00$00$00$00$00$00$00$00$00$00$00$00$00$00$00$00$00$00$00$00$00$00$00$00$00$00$00$00$00$00$00$00$00$00$00$00$00$00$00$00$00$00$00$00$00$00$00$00$00$00$00$00$00$00$14$00$00$007$01$00$00$00$00HB$00$00HB', HMI.Testing.Part[77].Results := 2046, HMI.Testing.Part[78].Code := '$00$00$00$00$8C$10$01$A02$00$00$002$00$00$00P$00$00$80$0C$00$00$80$04R9$F1$1C$12$D0$03$C2@@$00$01$00$00$00$00$00$00$00$03$00$00$007$01', HMI.Testing.Part[78].Results := 13, HMI.Testing.Part[80].Code := '010062810150300021T15UOB00031$0D$00$00$00$00$00$00$00$00$00$00$00$00$00$00$00$00$00$00$00$00$00$00$00$00$00$00$00$00$00$00$00$00$00$00$00$00$00$00$00$00$00$00$00$00$00$00$00$00$00$00$00$00$00$00', HMI.Testing.Part[80].Results := 20, HMI.Testing.Part[81].Code := '$00$00HB$00$00HB$FE$07$01$002$00$00$00$00$00$00$00$8C$10$01$A02$00$00$002$00$00$00P$00$00$80$0C$00$00$80$04R9$F1$1C$12$D0$03$C2@@$00$01$00$00$00$00$00$00$00$03$00$00$007$01$00$00$00$00HB$00$00HB$A7$0F$01$002$00$00$00', HMI.Testing.Part[82].Code := '2$00$00$00$DC$00$00$00$0D$00$00$00$00$00$00$00$00$00$00$00$08$00$00$80$1E$00$00$80$04R9$F1$14$13$D0$03$C2@>$00$01$00$00$00$1C$00$00$00$03$00$00$00$00$00$00$00$0B$00$00$00$00$00$CD$1CjAgf$E4A$CD$CCL$B9$CD$CCL$B9$00$00$00$00$00$00', HMI.Testing.Part[85].Code := '$A7$0F$01$002$00$00$00$00$00$00$00$8D$10$01$B12$00$00$00$DC$00$00$00$0D$00$00$00$00$00$00$00$00$00$00$00$08$00$00$80$1E$00$00$80$04R9$F1$14$13$D0$03$C2@>$00$01$00$00$00$1C$00$00$00$03$00$00$00$00$00$00$00$0B$00$00$00$00$00$CD$1CjAgf', HMI.Testing.Part[85].Results := 16868, HMI.Testing.Part[86].Code := 'L$B9$00$00$00$00$00$00$00$00$00$00$00$00$00$00$00$00$00$00$00$00$00$00$00$00$00$00ERRO010062810150300021T15UOB00031$0D$00$00$00$00$00$00$00$00$00$00$00$00$00$00$00$00$00$00$00$00$00$00', HMI.Testing.Part[87].Results := 1, HMI.Testing.Part[89].Code := '$00$00$CD$1CjAgf$E4A$CD', HMI.Testing.Part[90].Results := 12, HMI.Testing.Part[91].Code := '$1C$12$D0$03$C2@@$00$01$00$00$00$00$00$00$00$03$00$00$007$01$00$00$00$00HB$00$00HB$A7$0F$01$002$00$00$00$00$00$00$00$8D$10$01$B12$00$00$00$DC$00$00$00$0D$00$00$00$00$00$00$00$00$00$00$00$08$00$00$80$1E$00$00$80$04R9$F1$14$13$D0$03', HMI.Testing.Part[91].Results := 16578, HMI.Testing.Part[92].Code := '$1C', HMI.Testing.Part[92].Results := 21813, HMI.Testing.Part[93].Code := '1$0D$00$00$00$00$00$00$00$00$00$00$00$00$00$00$00$00$00$00$00$00$00$00$00$00$00$00$00$00$00$00$00$00$00$00$00$00$00$00$00$00$00$00$00$00$00$00$00$00$00$00$00$00$00$00$14$00$00$007$01$00$00$00$00HB$00$00HB$FE$07$01$002$00$00$00$00$00$00$00', HMI.Testing.Part[93].Results := 4236, HMI.Testing.Part[94].Code := '2$00$00$00P$00$00$80$0C$00$00$80$04R9$F1$1C$12$D0$03$C2@@$00$01$00$00$00$00$00$00$00$03$00$00$007$01$00$00$00$00HB$00$00HB$A7$0F', HMI.Testing.Part[94].Results := 8, HMI.Testing.Part[95].Code := '$04R9$F1$14$13$D0$03$C2@>$00$01$00$00$00$1C$00$00$00$03$00$00$00$00$00$00$00$0B$00$00$00$00$00$CD$1CjAgf$E4A$CD$CCL$B9$CD$CCL$B9$00$00$00$00$00$00$00$00$00$00$00$00$00$00$00$00$00$00$00$00$00$00$00$00$00$00ERRO0100', HMI.Testing.Part[95].Results := 12854, HMI.Testing.Part[96].Code := '300021T15UOB00031$0D$00$00$00$00$00$00$00$00$00$00$00$00$00$00$00$00$00$00$00$00$00$00$00$00$00$00$00$00$00$00$00$00$00$00$00$00$00$00$00$00$00$00$00$00$00$00$00$00$00$00$00$00$00$00$14$00$00$007$01$00$00$00$00HB', HMI.Testing.Part[97].Code := '2$00$00$00$00$00$00$00$8C$10$01$A02$00$00$002$00$00$00P$00$00$80$0C$00$00$80$04R9$F1$1C$12$D0$03$C2@@$00$01$00$00$00$00$00$00$00$03$00$00$007$01$00$00$00$00HB$00$00HB$A7$0F$01$002$00$00$00$00$00$00$00$8D$10$01$B12$00$00$00', HMI.Testing.Part[97].Results := 220, HMI.Testing.Part[98].Code := '$00$00$00$00$00$00$00$00$08$00$00$80$1E', HMI.Testing.Test[0].Flow := 2.8e-44, HMI.Testing.Test[0].Range := 4.36e-43, HMI.Testing.Test[0].Test_TM.PRE := 1112014848, HMI.Testing.Test[0].Test_TM.ACC := 67582, HMI.Testing.Test[0].Test_TM.TT := 1, HMI.Testing.Test[0].Time := 50, HMI.Testing.Test[1].Range := -1.09322e-19, HMI.Testing.Test[1].Test_TM.PRE := 50, HMI.Testing.Test[1].Test_TM.ACC := -2147483568, HMI.Testing.Test[1].Time := 12, HMI.Testing.Test[2].Flow := -9.1766204e+29, HMI.Testing.Test[2].Range := 1.2229299e-36, HMI.Testing.Test[2].Test_TM.PRE := 1, HMI.Testing.Test[2].Time := 3, HMI.Testing.Test[3].Flow := 4.36e-43, HMI.Testing.Test[3].Range := 50.0,
        HMI.Testing.Test[3].Test_TM.PRE := 69543, HMI.Testing.Test[3].Test_TM.ACC := 50, HMI.Testing.Test[3].Test_TM.TT := 1, HMI.Testing.Test[4].Flow := -1.8781379e-09, HMI.Testing.Test[4].Range := 7.e-44, HMI.Testing.Test[4].Test_TM.PRE := 13, HMI.Testing.Test[5].Flow := -1.1e-44, HMI.Testing.Test[5].Range := -4.2e-44, HMI.Testing.Test[5].Test_TM.PRE := 63968020, HMI.Testing.Test[5].Test_TM.ACC := 4079810, HMI.Testing.Test[5].Test_TM.EN := 1, HMI.Testing.Test[5].Test_TM.TT := 1, HMI.Testing.Test[5].Test_TM.DN := 1, HMI.Testing.Test[5].Time := 1, HMI.Testing.Test[6].Flow := 3.9e-44, HMI.Testing.Test[6].Range := 4.e-45, HMI.Testing.Test[6].Test_TM.PRE := 11, HMI.Testing.Test[6].Test_TM.ACC := 483196928, HMI.Testing.Test[6].Time := 16746, HMI.Testing.Load_PB.INPUT := 1, HMI.Testing.Load_PB.ON_TIME := -107858530.0, HMI.Testing.Load_PB.OFF_TIME := 6.6472e-41, HMI.Testing.Load_PB.IN := 1, HMI.Testing.Load_PB.ON_TT := 1, HMI.Testing.Load_PB.OFF_TT := 1, HMI.Testing.Load_PB.OUT := 1, HMI.Testing.Knob_Turner.Turn_Speed := 500.0, HMI.Testing.Knob_Turner.Rapid_Speed := 600.0, HMI.Testing.Knob_Turner.Torque1 := 45.0, HMI.Testing.Knob_Turner.Torque2 := 100.0, HMI.Part_Count := 808464688, HMI.Lifetime_Part_Count := 2.6804066e-09, HMI.Fault_AOI[0].Timer_PRE := 808464435, HMI.Fault_AOI[0].Timer_ACC := 827601202, HMI.Fault_AOI[0].Faulted := 1, HMI.Fault_AOI[0].Reset := 1, HMI.Fault_AOI[3].Timer_PRE := 20, HMI.Fault_AOI[3].Timer_ACC := 311, HMI.Fault_AOI[4].Timer_ACC := -1610542964, HMI.Fault_AOI[4].Faulted := 1, HMI.Fault_AOI[4].Reset := 1, HMI.Fault_AOI[5].Fault := 1, HMI.Fault_AOI[5].Bypass := 1, HMI.Fault_AOI[5].Timer_PRE := -247901692, HMI.Fault_AOI[5].Timer_ACC := 63967772, HMI.Fault_AOI[6].Timer_PRE := 311, HMI.Fault_AOI[6].Timer_ACC := 1112014848, HMI.Fault_AOI[7].Timer_PRE := -1325330291, HMI.Fault_AOI[7].Timer_ACC := 50, HMI.Fault_AOI[8].Timer_PRE := -2147483640, HMI.Fault_AOI[8].Timer_ACC := -2147483618, HMI.Fault_AOI[9].Timer_PRE := 28, HMI.Fault_AOI[9].Timer_ACC := 3, HMI.Fault_AOI[10].Bypass := 1, HMI.Fault_AOI[10].Timer_PRE := -858963484, HMI.Fault_AOI[10].Timer_ACC := -858932916, HMI.Fault_AOI[10].Reset := 1, HMI.Fault_AOI[12].Fault := 1, HMI.Fault_AOI[12].Timer_PRE := 808792368, HMI.Fault_AOI[12].Timer_ACC := 808464435,
        HMI.Fault_AOI[12].Faulted := 1, HMI.Fault_AOI[12].Reset := 1, HMI.Fault_AOI[13].Faulted := 1, HMI.Fault_AOI[13].Reset := 1, HMI.Fault_AOI[15].Timer_ACC := 20, HMI.Fault_AOI[16].Fault := 1, HMI.Fault_AOI[16].Bypass := 1, HMI.Fault_AOI[16].Timer_PRE := 50, HMI.Fault_AOI[16].Faulted := 1, HMI.Fault_AOI[16].Reset := 1, HMI.Fault_AOI[17].Timer_PRE := -2147483636, HMI.Fault_AOI[17].Timer_ACC := -247901692, HMI.Fault_AOI[17].Faulted := 1, HMI.Fault_AOI[18].Timer_PRE := 3, HMI.Fault_AOI[18].Timer_ACC := 311, HMI.Fault_AOI[19].Timer_ACC := -1325330291, HMI.Fault_AOI[19].Faulted := 1, HMI.Fault_AOI[19].Reset := 1, HMI.Fault_AOI[20].Timer_ACC := -2147483640, HMI.Fault_AOI[21].Timer_PRE := 1, HMI.Fault_AOI[21].Timer_ACC := 28, HMI.Fault_AOI[22].Timer_PRE := 1718042986, HMI.Fault_AOI[22].Timer_ACC := -858963484, HMI.Fault_AOI[24].Timer_PRE := 825766454, HMI.Fault_AOI[24].Timer_ACC := 808792368, HMI.Fault_AOI[24].Faulted := 1, HMI.Fault_AOI[24].Reset := 1, HMI.Fault_AOI[25].Timer_PRE := 3377, HMI.Fault_AOI[25].Faulted := 1, HMI.Fault_AOI[25].Reset := 1, HMI.Fault_AOI[28].Timer_PRE := 67582, HMI.Fault_AOI[28].Timer_ACC := 50, HMI.Fault_AOI[29].Timer_PRE := -2147483568, HMI.Fault_AOI[29].Timer_ACC := -2147483636, HMI.Fault_AOI[29].Faulted := 1, HMI.Fault_AOI[29].Reset := 1, HMI.Fault_AOI[30].Timer_ACC := 3, HMI.Fault_AOI[31].Fault := 1, HMI.Fault_AOI[31].Timer_PRE := 50, HMI.Fault_AOI[31].Reset := 1, HMI.Fault[0] := 13, HMI.FAULTED[1] := -2147483640, HMI.HMI.Reset_Faults := 1, HMI.Performance := 6.5917316e-10, HMI.UptimeSTM.PRE := 827601202, HMI.UptimeSTM.ACC := 1112495413, HMI.UptimeSTM.DN := 1, HMI.UptimeM.PRE := 3377, HMI.UptimeM.DN := 1, HMI.UptimeM.OV := 1, HMI.DowntimeH.ACC := 20, HMI.UptimeTM.PRE := 1112014848, HMI.UptimeTM.ACC := 1112014848, HMI.Batch_Count := 67582);
        .Conv.Lift.Stop.Present.DEB_INPUT   // Lift and locate pallet present
        .Conv.Stop[0].Release   // Operator Pallet Stop
        .Conv.Diverter.Present.DEB_INPUT   // Rejected
        .Conv.Stop[2].Release   // Infeed Pallet Stop
        .Conv.Stop[3].Release   // Reject Pallet Stop
        .Testing.Alicat[0].Ready   // Alicat ready
        .Testing.Alicat[0].Flow   // Averaged flow over 1 sec
        .Testing.Alicat[1].Ready   // Alicat ready
        .Testing.Part_Present.DEB_INPUT   // Part present
        .Conv.Stop[1].Release   // Lift & Locate Pallet Stop
        .Testing.FastTest.Extd.DEB_INPUT   // Fasttest extended
   MCP_00 : UDT_ID86 := (IN.M01_UR20_16DI_P.Data.Ch_03 := 1, IN.M01_UR20_16DI_P.Data.Ch_04 := 1, IN.M01_UR20_16DI_P.Data.Ch_06 := 1, IN.M01_UR20_16DI_P.Data.Ch_07 := 1, IN.M01_UR20_16DI_P.Data.Ch_08 := 1, IN.M01_UR20_16DI_P.Data.Ch_10 := 1, IN.M01_UR20_16DI_P.Data.Ch_13 := 1, IN.M01_UR20_16DI_P.Data.Ch_14 := 1, IN.M01_UR20_16DI_P.Diagnostic.ModTyp := 15, IN.M01_UR20_16DI_P.Diagnostic.ChTyp := 112, IN.M01_UR20_16DI_P.Diagnostic.Diag_US_3 := 7, IN.M01_UR20_16DI_P.Diagnostic.Diag_US_4 := 9, IN.M02_UR20_16DI_P.Diagnostic.ModTyp := 15, IN.M02_UR20_16DI_P.Diagnostic.ChTyp := 112, IN.M02_UR20_16DI_P.Diagnostic.Diag_US_3 := 7, IN.M02_UR20_16DI_P.Diagnostic.Diag_US_4 := 9, IN.M03_UR20_4AI_UI_16.Diagnostic.ModTyp := 5, IN.M03_UR20_4AI_UI_16.Diagnostic.ChTyp := 116, IN.M03_UR20_4AI_UI_16.Diagnostic.NumCh := 4, IN.M03_UR20_4AI_UI_16.Diagnostic.Diag_US_3 := 16, IN.M03_UR20_4AI_UI_16.Diagnostic.Diag_US_4 := 60, IN.M04_UR20_16DO_P.Diagnostic.ModTyp := 15, IN.M04_UR20_16DO_P.Diagnostic.ChTyp := 114, IN.M04_UR20_16DO_P.Diagnostic.Diag_US_3 := 7, IN.M04_UR20_16DO_P.Diagnostic.Diag_US_4 := 9, IN.M05_UR20_16DO_P.Diagnostic.ModTyp := 15, IN.M05_UR20_16DO_P.Diagnostic.ChTyp := 114, IN.M05_UR20_16DO_P.Diagnostic.Diag_US_3 := 7, IN.M05_UR20_16DO_P.Diagnostic.Diag_US_4 := 9, OUT.M04_UR20_16DO_P.Data.Ch_00 := 1, OUT.M04_UR20_16DO_P.Data.Ch_05 := 1, MISC.Startup_Flag := 1, MISC.Tmr_ProcessAlarm.PRE := 64, MISC.Tmr_ProcessAlarm.ACC := 30, MISC.Tmr_ProcessAlarm.EN := 1, MISC.Tmr_ProcessAlarm.TT := 1, MISC.Tmr_Diag.PRE := 64, MISC.Tmr_Diag.ACC := 30, MISC.Tmr_Diag.EN := 1, MISC.Tmr_Diag.TT := 1, MISC.Tmr_SetDefault.PRE := 200, MISC.DiagnosticData[1] := 15, MISC.DiagnosticData[4] := 114, MISC.DiagnosticData[45] := 7, MISC.DiagnosticData[46] := 9, MISC.InputBytes := 12, MISC.OutputBytes := 4, MISC.ParameterBytes := 17);
   Open : BOOL;
   Open_CMD : BOOL;
   Open_Go_ONS : BOOL;
   Open_ONS : BOOL;
   Open_ONS_CMD : BOOL;
   Open_Stop : BOOL;
   Open_Torque : INT := 36;
   Open_Torque_TMR : TIMER;
   Pallet_Release_TMR : TIMER := (PRE := 1600);
   Pallet_TMR : TIMER;
   Part_Delay : TIMER := (PRE := 2000);
   Part_Delay_2 : TIMER;
   PH_Cntr : COUNTER[5] := ([0].PRE := 100);
   PH_Cntr_ONS : BOOL;
   PH_Debug : DINT := 1413481728;
   PH_Debug_Tmr : TIMER[20] := ([0].PRE := 250, [1].PRE := 250, [2].PRE := 250, [3].PRE := 250, [4].PRE := 250, [5].PRE := 250, [6].PRE := 250, [6].ACC := 250, [6].EN := 1, [6].DN := 1, [7].PRE := 250, [8].PRE := 250, [9].PRE := 250, [10].PRE := 250, [11].PRE := 250, [12].PRE := 250, [13].PRE := 500);
   PH_ONS : INT;
   PH_Timer : TIMER[5] := ([0].PRE := 25000, [1].PRE := 500, [2].PRE := 500);
   RCP1 : RCP1 := (Inlet_Driver.Ret := 1, Inlet_Driver.Extd.ON_TIME := 50.0, Inlet_Driver.Extd.OFF_TIME := 50.0, Inlet_Driver.Retd.ON_TIME := 50.0, Inlet_Driver.Retd.OFF_TIME := 50.0, Inlet_Driver.Drive_TM.PRE := 1000, Needle_Driver.Ret := 1, Needle_Driver.Extd.ON_TIME := 50.0, Needle_Driver.Extd.OFF_TIME := 50.0, Needle_Driver.Retd.ON_TIME := 50.0, Needle_Driver.Retd.OFF_TIME := 50.0, Needle_Driver.Drive_TM.PRE := 1000, Saftey.Lockout := 1, Saftey.Estop := 1, Saftey.Light_Curtain := 1, Saftey.RDC_Code := 15233, Part_Present.ON_TIME := 50.0, Part_Present.OFF_TIME := 50.0, Part_Count := 74, Lifetime_Part_Count := 97.0, Home_PB.ON_TIME := 50.0, Home_PB.OFF_TIME := 50.0, Select_Switch.ON_TIME := 50.0, Select_Switch.OFF_TIME := 50.0, Reset_PB.ON_TIME := 50.0, Reset_PB.OFF_TIME := 50.0, Stacklight.Yellow := 1, Stacklight.Blue := 1, Fault_AOI[0].Timer_PRE := 10, Fault_AOI[1].Fault := 1, Fault_AOI[1].Timer_PRE := 10, Fault_AOI[1].Timer_ACC := 10, Fault_AOI[1].Faulted := 1, Fault_AOI[2].Timer_PRE := 1000, Fault_AOI[3].Fault := 1, Fault_AOI[3].Timer_PRE := 1000, Fault_AOI[3].Timer_ACC := 1000, Fault_AOI[3].Faulted := 1, Fault_AOI[4].Fault := 1, Fault_AOI[4].Timer_PRE := 100, Fault_AOI[4].Timer_ACC := 100, Fault_AOI[4].Faulted := 1, Fault_AOI[5].Fault := 1, Fault_AOI[5].Timer_PRE := 100, Fault_AOI[5].Timer_ACC := 100, Fault_AOI[5].Faulted := 1, Fault_AOI[6].Timer_PRE := 750, Fault_AOI[7].Timer_PRE := 750, Fault_AOI[8].Fault := 1, Fault_AOI[8].Timer_PRE := 750, Fault_AOI[8].Timer_ACC := 750, Fault_AOI[8].Faulted := 1, Fault_AOI[9].Timer_PRE := 750, Fault_AOI[10].Fault := 1, Fault_AOI[10].Timer_PRE := 750, Fault_AOI[10].Timer_ACC := 750, Fault_AOI[10].Faulted := 1, Fault := 1338, FAULTED := 1338, Air_Pressure.ON_TIME := 50.0,
        Air_Pressure.OFF_TIME := 50.0, HMI.Max_Cycle_Time := 25.0, Max_Cycle_Time := 25, Performance := inf, Availability := inf, UptimeTM.PRE := 1000, UptimeS.PRE := 60, UptimeM.PRE := 60, UptimeH.DN := 1, DowntimeTM.PRE := 1000, DowntimeTM.ACC := 300, DowntimeTM.EN := 1, DowntimeTM.TT := 1, DowntimeS.PRE := 60, DowntimeS.ACC := 14, DowntimeM.PRE := 60, DowntimeM.ACC := 6, DowntimeH.ACC := 22, DowntimeH.DN := 1, Batch_Count := 70);
        .Inlet_Driver.Extd   // Inlet Driver Cylinder Extended
        .Needle_Driver.Retd   // Needle Driver Cylinder Retracted
        .Part_Present   // Part present
        .Needle_Driver.Extd   // Needle Driver Cylinder Extended
        .Inlet_Driver.Retd   // Inlet Driver Cylinder Retracted
   RCP1_00 : UDT_ID0 := (IN.M01_UR20_16DI_P.Diagnostic.ModTyp := 15, IN.M01_UR20_16DI_P.Diagnostic.ChTyp := 112, IN.M01_UR20_16DI_P.Diagnostic.Diag_US_3 := 5, IN.M01_UR20_16DI_P.Diagnostic.Diag_US_4 := -89, IN.M02_UR20_16DI_P.Diagnostic.ModTyp := 15, IN.M02_UR20_16DI_P.Diagnostic.ChTyp := 112, IN.M02_UR20_16DI_P.Diagnostic.Diag_US_3 := 5, IN.M02_UR20_16DI_P.Diagnostic.Diag_US_4 := -89, IN.M03_UR20_4AI_UI_16.Diagnostic.ModTyp := 5, IN.M03_UR20_4AI_UI_16.Diagnostic.ChTyp := 116, IN.M03_UR20_4AI_UI_16.Diagnostic.NumCh := 4, IN.M03_UR20_4AI_UI_16.Diagnostic.Diag_US_3 := 16, IN.M03_UR20_4AI_UI_16.Diagnostic.Diag_US_4 := 60, IN.M04_UR20_16DO_P.Diagnostic.ModTyp := 15, IN.M04_UR20_16DO_P.Diagnostic.ChTyp := 114, IN.M04_UR20_16DO_P.Diagnostic.Diag_US_3 := 7, IN.M04_UR20_16DO_P.Diagnostic.Diag_US_4 := 9, IN.M05_UR20_16DO_P.Diagnostic.ModTyp := 15, IN.M05_UR20_16DO_P.Diagnostic.ChTyp := 114, IN.M05_UR20_16DO_P.Diagnostic.Diag_US_3 := 7, IN.M05_UR20_16DO_P.Diagnostic.Diag_US_4 := 9, OUT.M04_UR20_16DO_P.Data.Ch_03 := 1, MISC.Startup_Flag := 1, MISC.Tmr_ProcessAlarm.PRE := 64, MISC.Tmr_Diag.PRE := 64, MISC.Tmr_SetDefault.PRE := 200, MISC.DiagnosticData[1] := 15, MISC.DiagnosticData[4] := 112, MISC.DiagnosticData[45] := 5, MISC.DiagnosticData[46] := -89, MISC.InputBytes := 12, MISC.OutputBytes := 4, MISC.ParameterBytes := 17);
   Read_Barcode_ONS : BOOL;
   Reject : BOOL;
   Reject_Active : BOOL;
   Reject_Barcode : BOOL;
   Reject_CTR : COUNTER := (PRE := 10000, ACC := 11);
   Reject_Delay : BOOL;
   Reject_Delay_TMR : TIMER := (PRE := 3000);
   Reject_ONS : BOOL;
   Reject_Pallet : BOOL := 1;
   Reject_Pallet1_ONS : BOOL;
   Reject_Pallet_Bit : DINT;
        .1   // Leak Test
        .2   // 8LPM Test
        .5   // 2LPM Test
        .3   // 15LPM Test
        .4   // Flood Test
   Reject_Pallet_ONS : BOOL;
   Reject_Pallets_TMR : TIMER := (PRE := 5000, ACC := 1600, EN := 1, TT := 1);
   Reject_TMR : TIMER;
   Reset_ONS : BOOL;
   Rotation_Cycles : INT := 1;
   Safety_OK : BOOL := 1;
   Temp_Cycle_Time : INT := -30906;
   Temp_Cycle_Time_Current : REAL := 2.05;
   Temp_Cycle_Time_DINT : DINT := 43170;
   Temp_Cycle_Time_Last : REAL := 3.38;
   Temp_Cycle_Timer : TIMER := (PRE := 999999, ACC := 2050);
   Temp_Cycle_Timer_BIT : BOOL;
   Temp_Cycle_Timer_ONF : BOOL := 1;
   Test2_Rapid : Servo_Move := (Speed := 600.0, Torque := 100.0, Position := -25000.0, Path := 1);
   Test2_Step : Servo_Move := (Speed := 100.0, Torque := 45.0, Position := 250000.0, Path := 1);
   Test3_Rapid : Servo_Move := (Speed := 1000.0, Torque := 100.0, Path := 1);
   Test3_Step : Servo_Move := (Speed := 200.0, Torque := 100.0, Position := -600000.0, Path := 1);
   Test4_Rapid : Servo_Move := (Speed := 1000.0, Torque := 100.0, Position := -45000.0, Path := 1);
   Test4_Step : Servo_Move := (Speed := 200.0, Torque := 100.0, Position := -600000.0, Path := 1);
   Test5_Rapid : Servo_Move := (Speed := 2000.0, Torque := 60.0, Position := -25000.0, Path := 1);
   Test5_Step : Servo_Move := (Speed := 1000.0, Torque := 45.0, Position := -4000000.0, Path := 1);
   Test_Close : Servo_Move := (Speed := 800.0, Torque := 45.0, Position := 1000000.0);
   Test_Close_nudge : Servo_Move := (Speed := 600.0, Torque := 80.0, Position := 10000.0);
   Test_Close_Rapid : Servo_Move := (Speed := 6000.0, Torque := 99.0, Position := 400000.0);
   Test_Data : REAL[8] := ([1] := 0.0001953125, [2] := 6.9492188, [3] := 15.0859375, [4] := 52.21875, [5] := 0.0005859375);
   Test_Data_Moved : BOOL;
   Test_Data_ONS : BOOL[32];
   Test_Delay_TMR : TIMER[5] := ([0].PRE := 1000, [1].PRE := 1000, [2].PRE := 1000, [3].PRE := 1000, [4].PRE := 1000);
   Test_Open : Servo_Move := (Speed := 800.0, Torque := 45.0, Position := -1000000.0);
   Test_Open_Rapid : Servo_Move := (Speed := 6000.0, Torque := 99.0, Position := -400000.0, DN := 1);
   Torque : DINT := 43;
   Torque_Start_TM : TIMER[2] := ([0].PRE := 1500, [1].PRE := 1500);
   Transmit_Data : BOOL := 1;
   Trig_Path_ONS : BOOL[32];
   Trig_Path_TM : TIMER[2] := ([0].PRE := 100, [1].PRE := 200);
   Vision_Result_OK_TMR : TIMER[6] := ([2].PRE := 500, [3].PRE := 500, [5].PRE := 500);
   Vision_TMR : TIMER[3] := ([0].PRE := 1000, [1].PRE := 1000, [2].PRE := 1000);
   Zero_Data : Servo_Move := (Torque := 100.0, Path := 1);
END_VAR
